// Mitsubishi GX Developer project: 粗材ストッカー   PLC: Q02

PROGRAM MAIN
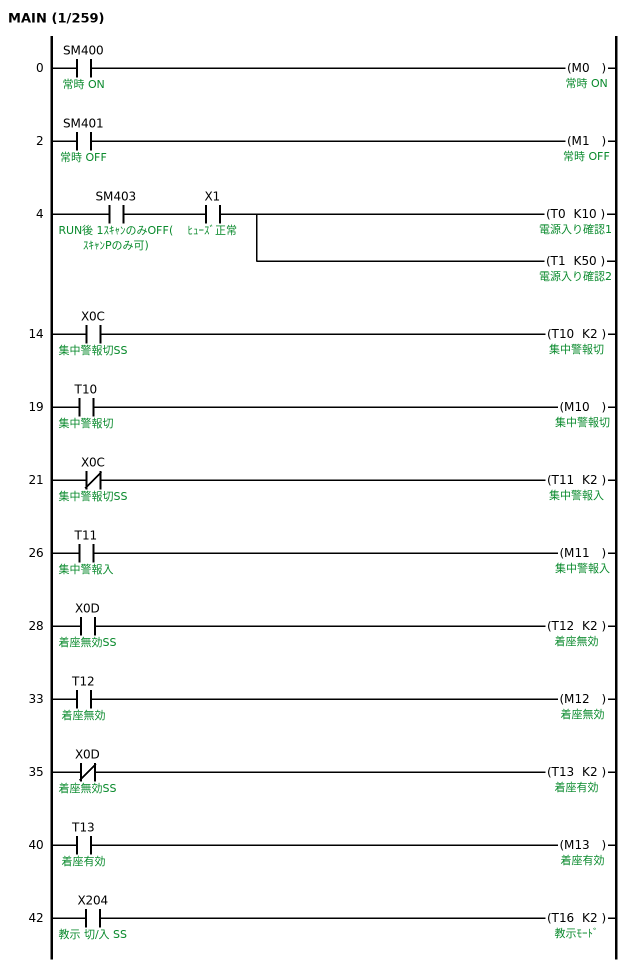
0     LD      SM400  ; 常時 ON
      OUT     M0  ; 常時 ON
2     LD      SM401  ; 常時 OFF
      OUT     M1  ; 常時 OFF
4     LD      SM403  ; RUN後 1ｽｷｬﾝのみOFF(ｽｷｬﾝPのみ可)
      AND     X1  ; ﾋｭｰｽﾞ正常
      OUT     T0 K10  ; 電源入り確認1
      OUT     T1 K50  ; 電源入り確認2
14    LD      X0C  ; 集中警報切SS
      OUT     T10 K2  ; 集中警報切
19    LD      T10  ; 集中警報切
      OUT     M10  ; 集中警報切
21    LDI     X0C  ; 集中警報切SS
      OUT     T11 K2  ; 集中警報入
26    LD      T11  ; 集中警報入
      OUT     M11  ; 集中警報入
28    LD      X0D  ; 着座無効SS
      OUT     T12 K2  ; 着座無効
33    LD      T12  ; 着座無効
      OUT     M12  ; 着座無効
35    LDI     X0D  ; 着座無効SS
      OUT     T13 K2  ; 着座有効
40    LD      T13  ; 着座有効
      OUT     M13  ; 着座有効
42    LD      X204  ; 教示 切/入 SS
      OUT     T16 K2  ; 教示ﾓｰﾄﾞ
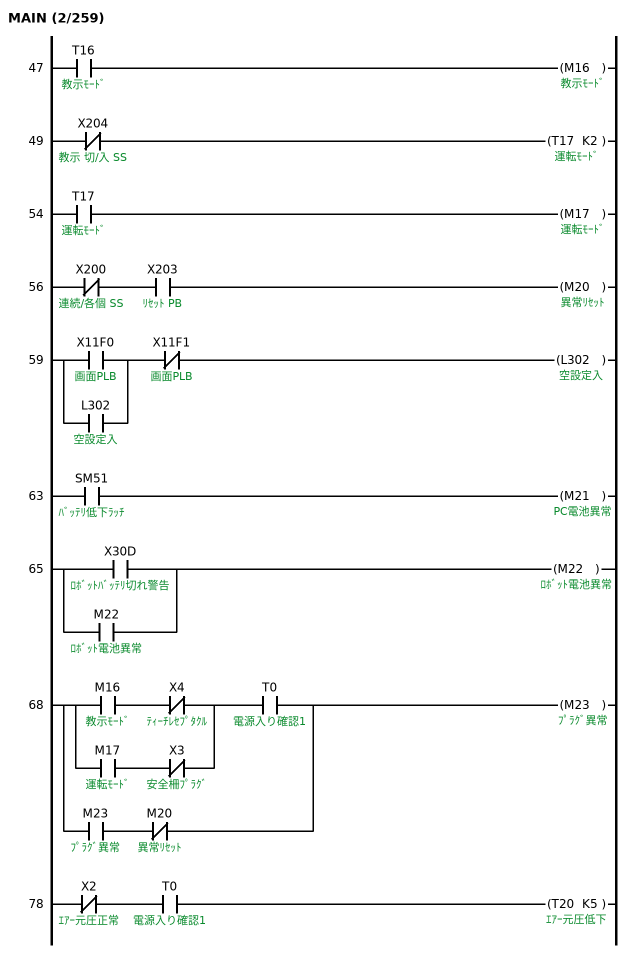
47    LD      T16  ; 教示ﾓｰﾄﾞ
      OUT     M16  ; 教示ﾓｰﾄﾞ
49    LDI     X204  ; 教示 切/入 SS
      OUT     T17 K2  ; 運転ﾓｰﾄﾞ
54    LD      T17  ; 運転ﾓｰﾄﾞ
      OUT     M17  ; 運転ﾓｰﾄﾞ
56    LDI     X200  ; 連続/各個 SS
      AND     X203  ; ﾘｾｯﾄ PB
      OUT     M20  ; 異常ﾘｾｯﾄ
59    LD      X11F0  ; 画面PLB
      OR      L302  ; 空設定入
      ANI     X11F1  ; 画面PLB
      OUT     L302  ; 空設定入
63    LD      SM51  ; ﾊﾞｯﾃﾘ低下ﾗｯﾁ
      OUT     M21  ; PC電池異常
65    LD      X30D  ; ﾛﾎﾞｯﾄﾊﾞｯﾃﾘ切れ警告
      OR      M22  ; ﾛﾎﾞｯﾄ電池異常
      OUT     M22  ; ﾛﾎﾞｯﾄ電池異常
68    LD      M16  ; 教示ﾓｰﾄﾞ
      ANI     X4  ; ﾃｨｰﾁﾚｾﾌﾟﾀｸﾙ
      LD      M17  ; 運転ﾓｰﾄﾞ
      ANI     X3  ; 安全柵ﾌﾟﾗｸﾞ
      ORB
      AND     T0  ; 電源入り確認1
      LD      M23  ; ﾌﾟﾗｸﾞ異常
      ANI     M20  ; 異常ﾘｾｯﾄ
      ORB
      OUT     M23  ; ﾌﾟﾗｸﾞ異常
78    LDI     X2  ; ｴｱｰ元圧正常
      AND     T0  ; 電源入り確認1
      OUT     T20 K5  ; ｴｱｰ元圧低下
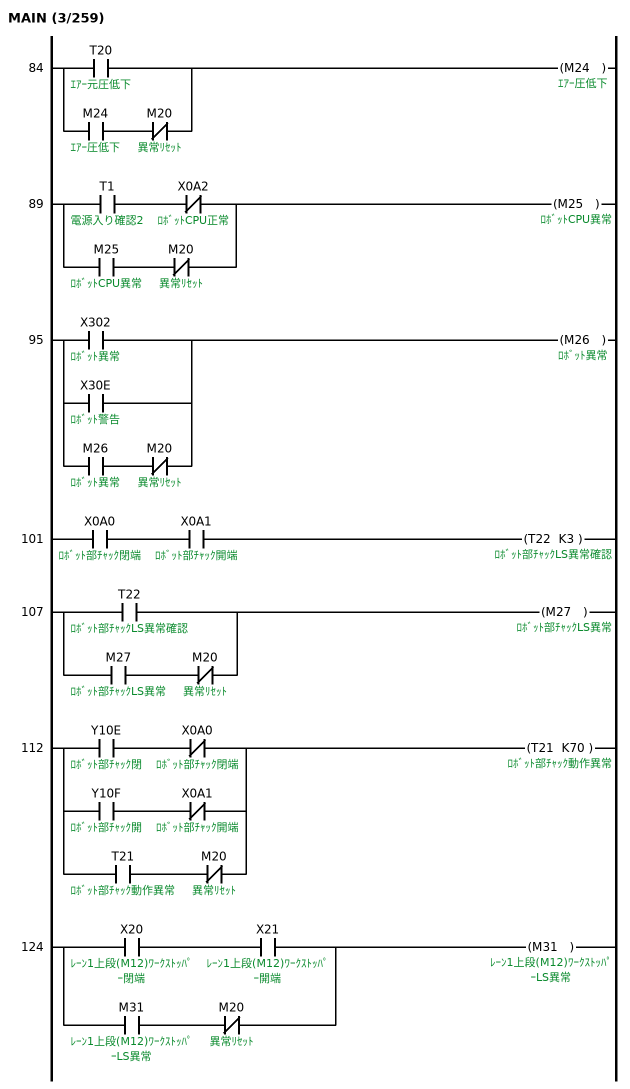
84    LD      T20  ; ｴｱｰ元圧低下
      LD      M24  ; ｴｱｰ圧低下
      ANI     M20  ; 異常ﾘｾｯﾄ
      ORB
      OUT     M24  ; ｴｱｰ圧低下
89    LD      T1  ; 電源入り確認2
      ANI     X0A2  ; ﾛﾎﾞｯﾄCPU正常
      LD      M25  ; ﾛﾎﾞｯﾄCPU異常
      ANI     M20  ; 異常ﾘｾｯﾄ
      ORB
      OUT     M25  ; ﾛﾎﾞｯﾄCPU異常
95    LD      X302  ; ﾛﾎﾞｯﾄ異常
      OR      X30E  ; ﾛﾎﾞｯﾄ警告
      LD      M26  ; ﾛﾎﾞｯﾄ異常
      ANI     M20  ; 異常ﾘｾｯﾄ
      ORB
      OUT     M26  ; ﾛﾎﾞｯﾄ異常
101   LD      X0A0  ; ﾛﾎﾞｯﾄ部ﾁｬｯｸ閉端
      AND     X0A1  ; ﾛﾎﾞｯﾄ部ﾁｬｯｸ開端
      OUT     T22 K3  ; ﾛﾎﾞｯﾄ部ﾁｬｯｸLS異常確認
107   LD      T22  ; ﾛﾎﾞｯﾄ部ﾁｬｯｸLS異常確認
      LD      M27  ; ﾛﾎﾞｯﾄ部ﾁｬｯｸLS異常
      ANI     M20  ; 異常ﾘｾｯﾄ
      ORB
      OUT     M27  ; ﾛﾎﾞｯﾄ部ﾁｬｯｸLS異常
112   LD      Y10E  ; ﾛﾎﾞｯﾄ部ﾁｬｯｸ閉
      ANI     X0A0  ; ﾛﾎﾞｯﾄ部ﾁｬｯｸ閉端
      LD      Y10F  ; ﾛﾎﾞｯﾄ部ﾁｬｯｸ開
      ANI     X0A1  ; ﾛﾎﾞｯﾄ部ﾁｬｯｸ開端
      ORB
      LD      T21  ; ﾛﾎﾞｯﾄ部ﾁｬｯｸ動作異常
      ANI     M20  ; 異常ﾘｾｯﾄ
      ORB
      OUT     T21 K70  ; ﾛﾎﾞｯﾄ部ﾁｬｯｸ動作異常
124   LD      X20  ; ﾚｰﾝ1上段(M12)ﾜｰｸｽﾄｯﾊﾟｰ閉端
      AND     X21  ; ﾚｰﾝ1上段(M12)ﾜｰｸｽﾄｯﾊﾟｰ開端
      LD      M31  ; ﾚｰﾝ1上段(M12)ﾜｰｸｽﾄｯﾊﾟｰLS異常
      ANI     M20  ; 異常ﾘｾｯﾄ
      ORB
      OUT     M31  ; ﾚｰﾝ1上段(M12)ﾜｰｸｽﾄｯﾊﾟｰLS異常
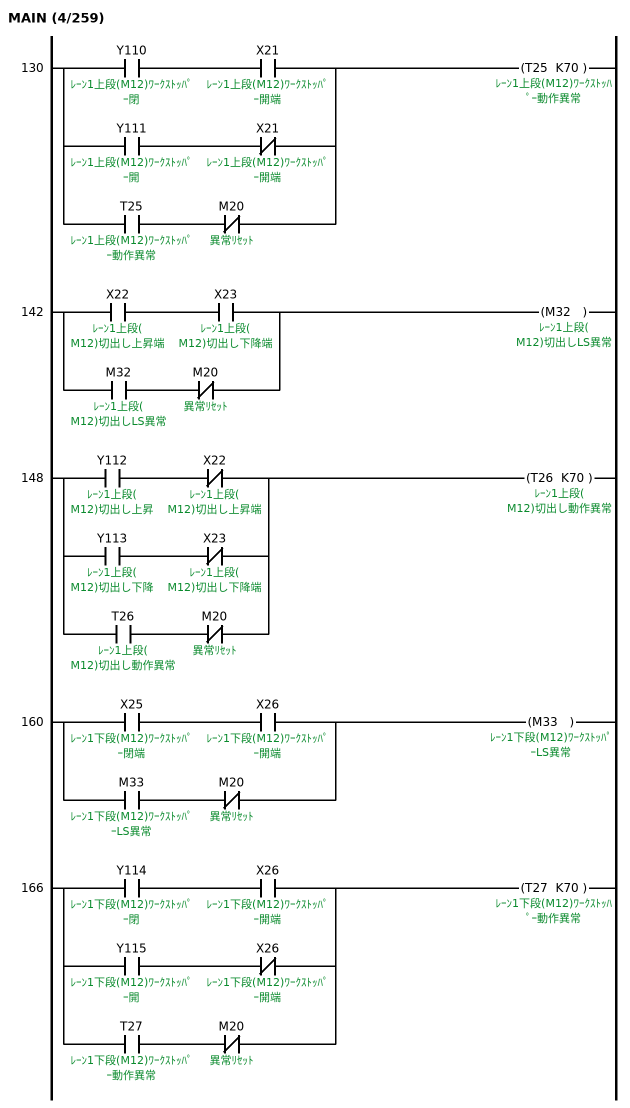
130   LD      Y110  ; ﾚｰﾝ1上段(M12)ﾜｰｸｽﾄｯﾊﾟｰ閉
      AND     X21  ; ﾚｰﾝ1上段(M12)ﾜｰｸｽﾄｯﾊﾟｰ開端
      LD      Y111  ; ﾚｰﾝ1上段(M12)ﾜｰｸｽﾄｯﾊﾟｰ開
      ANI     X21  ; ﾚｰﾝ1上段(M12)ﾜｰｸｽﾄｯﾊﾟｰ開端
      ORB
      LD      T25  ; ﾚｰﾝ1上段(M12)ﾜｰｸｽﾄｯﾊﾟｰ動作異常
      ANI     M20  ; 異常ﾘｾｯﾄ
      ORB
      OUT     T25 K70  ; ﾚｰﾝ1上段(M12)ﾜｰｸｽﾄｯﾊﾟｰ動作異常
142   LD      X22  ; ﾚｰﾝ1上段(M12)切出し上昇端
      AND     X23  ; ﾚｰﾝ1上段(M12)切出し下降端
      LD      M32  ; ﾚｰﾝ1上段(M12)切出しLS異常
      ANI     M20  ; 異常ﾘｾｯﾄ
      ORB
      OUT     M32  ; ﾚｰﾝ1上段(M12)切出しLS異常
148   LD      Y112  ; ﾚｰﾝ1上段(M12)切出し上昇
      ANI     X22  ; ﾚｰﾝ1上段(M12)切出し上昇端
      LD      Y113  ; ﾚｰﾝ1上段(M12)切出し下降
      ANI     X23  ; ﾚｰﾝ1上段(M12)切出し下降端
      ORB
      LD      T26  ; ﾚｰﾝ1上段(M12)切出し動作異常
      ANI     M20  ; 異常ﾘｾｯﾄ
      ORB
      OUT     T26 K70  ; ﾚｰﾝ1上段(M12)切出し動作異常
160   LD      X25  ; ﾚｰﾝ1下段(M12)ﾜｰｸｽﾄｯﾊﾟｰ閉端
      AND     X26  ; ﾚｰﾝ1下段(M12)ﾜｰｸｽﾄｯﾊﾟｰ開端
      LD      M33  ; ﾚｰﾝ1下段(M12)ﾜｰｸｽﾄｯﾊﾟｰLS異常
      ANI     M20  ; 異常ﾘｾｯﾄ
      ORB
      OUT     M33  ; ﾚｰﾝ1下段(M12)ﾜｰｸｽﾄｯﾊﾟｰLS異常
166   LD      Y114  ; ﾚｰﾝ1下段(M12)ﾜｰｸｽﾄｯﾊﾟｰ閉
      AND     X26  ; ﾚｰﾝ1下段(M12)ﾜｰｸｽﾄｯﾊﾟｰ開端
      LD      Y115  ; ﾚｰﾝ1下段(M12)ﾜｰｸｽﾄｯﾊﾟｰ開
      ANI     X26  ; ﾚｰﾝ1下段(M12)ﾜｰｸｽﾄｯﾊﾟｰ開端
      ORB
      LD      T27  ; ﾚｰﾝ1下段(M12)ﾜｰｸｽﾄｯﾊﾟｰ動作異常
      ANI     M20  ; 異常ﾘｾｯﾄ
      ORB
      OUT     T27 K70  ; ﾚｰﾝ1下段(M12)ﾜｰｸｽﾄｯﾊﾟｰ動作異常
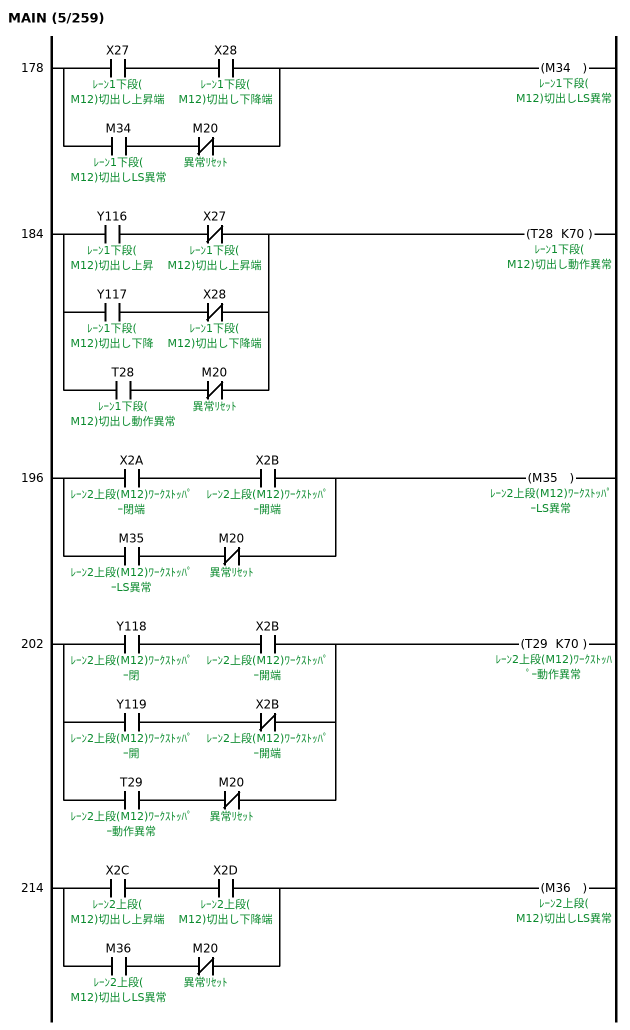
178   LD      X27  ; ﾚｰﾝ1下段(M12)切出し上昇端
      AND     X28  ; ﾚｰﾝ1下段(M12)切出し下降端
      LD      M34  ; ﾚｰﾝ1下段(M12)切出しLS異常
      ANI     M20  ; 異常ﾘｾｯﾄ
      ORB
      OUT     M34  ; ﾚｰﾝ1下段(M12)切出しLS異常
184   LD      Y116  ; ﾚｰﾝ1下段(M12)切出し上昇
      ANI     X27  ; ﾚｰﾝ1下段(M12)切出し上昇端
      LD      Y117  ; ﾚｰﾝ1下段(M12)切出し下降
      ANI     X28  ; ﾚｰﾝ1下段(M12)切出し下降端
      ORB
      LD      T28  ; ﾚｰﾝ1下段(M12)切出し動作異常
      ANI     M20  ; 異常ﾘｾｯﾄ
      ORB
      OUT     T28 K70  ; ﾚｰﾝ1下段(M12)切出し動作異常
196   LD      X2A  ; ﾚｰﾝ2上段(M12)ﾜｰｸｽﾄｯﾊﾟｰ閉端
      AND     X2B  ; ﾚｰﾝ2上段(M12)ﾜｰｸｽﾄｯﾊﾟｰ開端
      LD      M35  ; ﾚｰﾝ2上段(M12)ﾜｰｸｽﾄｯﾊﾟｰLS異常
      ANI     M20  ; 異常ﾘｾｯﾄ
      ORB
      OUT     M35  ; ﾚｰﾝ2上段(M12)ﾜｰｸｽﾄｯﾊﾟｰLS異常
202   LD      Y118  ; ﾚｰﾝ2上段(M12)ﾜｰｸｽﾄｯﾊﾟｰ閉
      AND     X2B  ; ﾚｰﾝ2上段(M12)ﾜｰｸｽﾄｯﾊﾟｰ開端
      LD      Y119  ; ﾚｰﾝ2上段(M12)ﾜｰｸｽﾄｯﾊﾟｰ開
      ANI     X2B  ; ﾚｰﾝ2上段(M12)ﾜｰｸｽﾄｯﾊﾟｰ開端
      ORB
      LD      T29  ; ﾚｰﾝ2上段(M12)ﾜｰｸｽﾄｯﾊﾟｰ動作異常
      ANI     M20  ; 異常ﾘｾｯﾄ
      ORB
      OUT     T29 K70  ; ﾚｰﾝ2上段(M12)ﾜｰｸｽﾄｯﾊﾟｰ動作異常
214   LD      X2C  ; ﾚｰﾝ2上段(M12)切出し上昇端
      AND     X2D  ; ﾚｰﾝ2上段(M12)切出し下降端
      LD      M36  ; ﾚｰﾝ2上段(M12)切出しLS異常
      ANI     M20  ; 異常ﾘｾｯﾄ
      ORB
      OUT     M36  ; ﾚｰﾝ2上段(M12)切出しLS異常
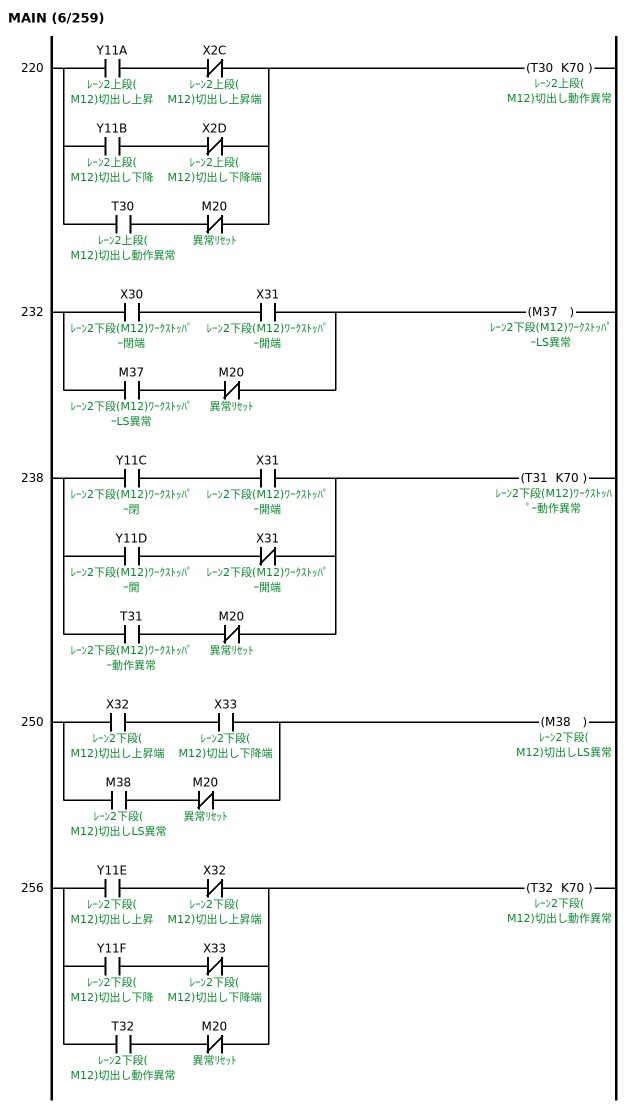
220   LD      Y11A  ; ﾚｰﾝ2上段(M12)切出し上昇
      ANI     X2C  ; ﾚｰﾝ2上段(M12)切出し上昇端
      LD      Y11B  ; ﾚｰﾝ2上段(M12)切出し下降
      ANI     X2D  ; ﾚｰﾝ2上段(M12)切出し下降端
      ORB
      LD      T30  ; ﾚｰﾝ2上段(M12)切出し動作異常
      ANI     M20  ; 異常ﾘｾｯﾄ
      ORB
      OUT     T30 K70  ; ﾚｰﾝ2上段(M12)切出し動作異常
232   LD      X30  ; ﾚｰﾝ2下段(M12)ﾜｰｸｽﾄｯﾊﾟｰ閉端
      AND     X31  ; ﾚｰﾝ2下段(M12)ﾜｰｸｽﾄｯﾊﾟｰ開端
      LD      M37  ; ﾚｰﾝ2下段(M12)ﾜｰｸｽﾄｯﾊﾟｰLS異常
      ANI     M20  ; 異常ﾘｾｯﾄ
      ORB
      OUT     M37  ; ﾚｰﾝ2下段(M12)ﾜｰｸｽﾄｯﾊﾟｰLS異常
238   LD      Y11C  ; ﾚｰﾝ2下段(M12)ﾜｰｸｽﾄｯﾊﾟｰ閉
      AND     X31  ; ﾚｰﾝ2下段(M12)ﾜｰｸｽﾄｯﾊﾟｰ開端
      LD      Y11D  ; ﾚｰﾝ2下段(M12)ﾜｰｸｽﾄｯﾊﾟｰ開
      ANI     X31  ; ﾚｰﾝ2下段(M12)ﾜｰｸｽﾄｯﾊﾟｰ開端
      ORB
      LD      T31  ; ﾚｰﾝ2下段(M12)ﾜｰｸｽﾄｯﾊﾟｰ動作異常
      ANI     M20  ; 異常ﾘｾｯﾄ
      ORB
      OUT     T31 K70  ; ﾚｰﾝ2下段(M12)ﾜｰｸｽﾄｯﾊﾟｰ動作異常
250   LD      X32  ; ﾚｰﾝ2下段(M12)切出し上昇端
      AND     X33  ; ﾚｰﾝ2下段(M12)切出し下降端
      LD      M38  ; ﾚｰﾝ2下段(M12)切出しLS異常
      ANI     M20  ; 異常ﾘｾｯﾄ
      ORB
      OUT     M38  ; ﾚｰﾝ2下段(M12)切出しLS異常
256   LD      Y11E  ; ﾚｰﾝ2下段(M12)切出し上昇
      ANI     X32  ; ﾚｰﾝ2下段(M12)切出し上昇端
      LD      Y11F  ; ﾚｰﾝ2下段(M12)切出し下降
      ANI     X33  ; ﾚｰﾝ2下段(M12)切出し下降端
      ORB
      LD      T32  ; ﾚｰﾝ2下段(M12)切出し動作異常
      ANI     M20  ; 異常ﾘｾｯﾄ
      ORB
      OUT     T32 K70  ; ﾚｰﾝ2下段(M12)切出し動作異常
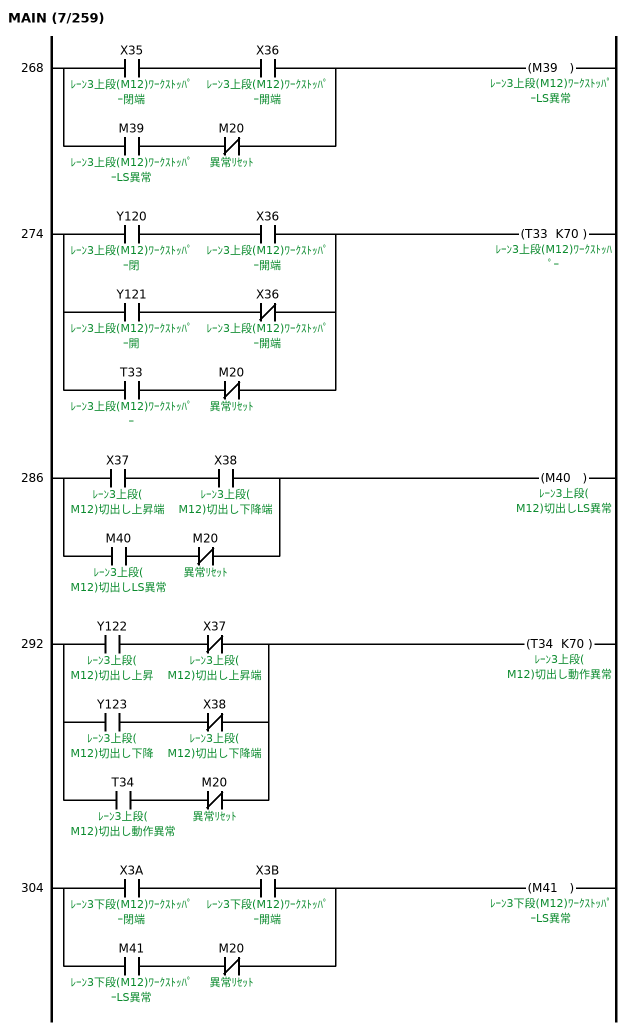
268   LD      X35  ; ﾚｰﾝ3上段(M12)ﾜｰｸｽﾄｯﾊﾟｰ閉端
      AND     X36  ; ﾚｰﾝ3上段(M12)ﾜｰｸｽﾄｯﾊﾟｰ開端
      LD      M39  ; ﾚｰﾝ3上段(M12)ﾜｰｸｽﾄｯﾊﾟｰLS異常
      ANI     M20  ; 異常ﾘｾｯﾄ
      ORB
      OUT     M39  ; ﾚｰﾝ3上段(M12)ﾜｰｸｽﾄｯﾊﾟｰLS異常
274   LD      Y120  ; ﾚｰﾝ3上段(M12)ﾜｰｸｽﾄｯﾊﾟｰ閉
      AND     X36  ; ﾚｰﾝ3上段(M12)ﾜｰｸｽﾄｯﾊﾟｰ開端
      LD      Y121  ; ﾚｰﾝ3上段(M12)ﾜｰｸｽﾄｯﾊﾟｰ開
      ANI     X36  ; ﾚｰﾝ3上段(M12)ﾜｰｸｽﾄｯﾊﾟｰ開端
      ORB
      LD      T33  ; ﾚｰﾝ3上段(M12)ﾜｰｸｽﾄｯﾊﾟｰ
      ANI     M20  ; 異常ﾘｾｯﾄ
      ORB
      OUT     T33 K70  ; ﾚｰﾝ3上段(M12)ﾜｰｸｽﾄｯﾊﾟｰ
286   LD      X37  ; ﾚｰﾝ3上段(M12)切出し上昇端
      AND     X38  ; ﾚｰﾝ3上段(M12)切出し下降端
      LD      M40  ; ﾚｰﾝ3上段(M12)切出しLS異常
      ANI     M20  ; 異常ﾘｾｯﾄ
      ORB
      OUT     M40  ; ﾚｰﾝ3上段(M12)切出しLS異常
292   LD      Y122  ; ﾚｰﾝ3上段(M12)切出し上昇
      ANI     X37  ; ﾚｰﾝ3上段(M12)切出し上昇端
      LD      Y123  ; ﾚｰﾝ3上段(M12)切出し下降
      ANI     X38  ; ﾚｰﾝ3上段(M12)切出し下降端
      ORB
      LD      T34  ; ﾚｰﾝ3上段(M12)切出し動作異常
      ANI     M20  ; 異常ﾘｾｯﾄ
      ORB
      OUT     T34 K70  ; ﾚｰﾝ3上段(M12)切出し動作異常
304   LD      X3A  ; ﾚｰﾝ3下段(M12)ﾜｰｸｽﾄｯﾊﾟｰ閉端
      AND     X3B  ; ﾚｰﾝ3下段(M12)ﾜｰｸｽﾄｯﾊﾟｰ開端
      LD      M41  ; ﾚｰﾝ3下段(M12)ﾜｰｸｽﾄｯﾊﾟｰLS異常
      ANI     M20  ; 異常ﾘｾｯﾄ
      ORB
      OUT     M41  ; ﾚｰﾝ3下段(M12)ﾜｰｸｽﾄｯﾊﾟｰLS異常
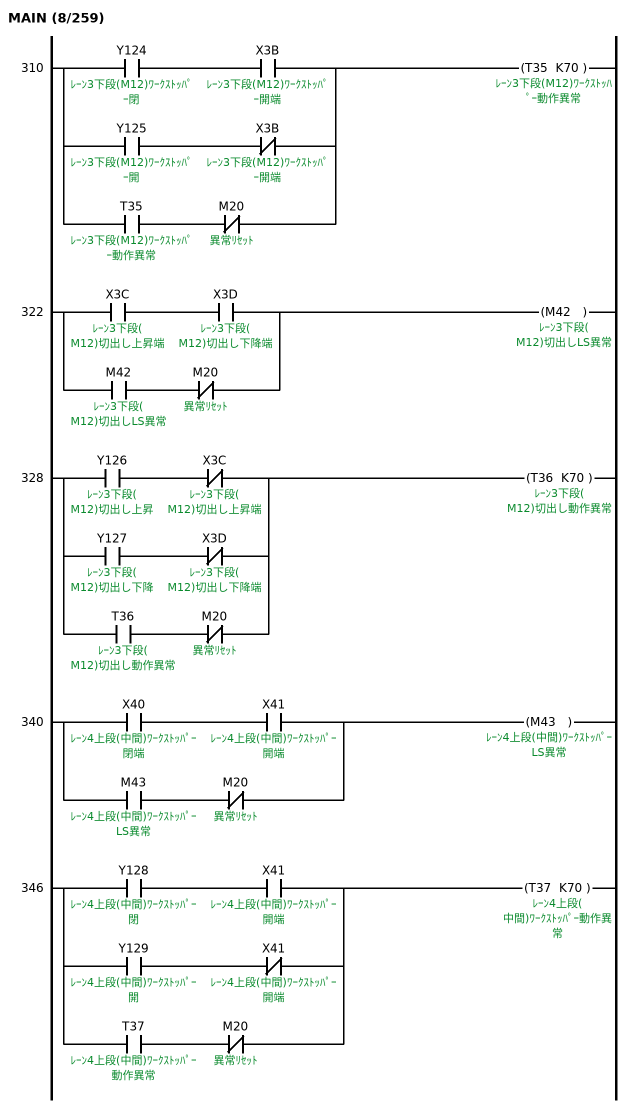
310   LD      Y124  ; ﾚｰﾝ3下段(M12)ﾜｰｸｽﾄｯﾊﾟｰ閉
      AND     X3B  ; ﾚｰﾝ3下段(M12)ﾜｰｸｽﾄｯﾊﾟｰ開端
      LD      Y125  ; ﾚｰﾝ3下段(M12)ﾜｰｸｽﾄｯﾊﾟｰ開
      ANI     X3B  ; ﾚｰﾝ3下段(M12)ﾜｰｸｽﾄｯﾊﾟｰ開端
      ORB
      LD      T35  ; ﾚｰﾝ3下段(M12)ﾜｰｸｽﾄｯﾊﾟｰ動作異常
      ANI     M20  ; 異常ﾘｾｯﾄ
      ORB
      OUT     T35 K70  ; ﾚｰﾝ3下段(M12)ﾜｰｸｽﾄｯﾊﾟｰ動作異常
322   LD      X3C  ; ﾚｰﾝ3下段(M12)切出し上昇端
      AND     X3D  ; ﾚｰﾝ3下段(M12)切出し下降端
      LD      M42  ; ﾚｰﾝ3下段(M12)切出しLS異常
      ANI     M20  ; 異常ﾘｾｯﾄ
      ORB
      OUT     M42  ; ﾚｰﾝ3下段(M12)切出しLS異常
328   LD      Y126  ; ﾚｰﾝ3下段(M12)切出し上昇
      ANI     X3C  ; ﾚｰﾝ3下段(M12)切出し上昇端
      LD      Y127  ; ﾚｰﾝ3下段(M12)切出し下降
      ANI     X3D  ; ﾚｰﾝ3下段(M12)切出し下降端
      ORB
      LD      T36  ; ﾚｰﾝ3下段(M12)切出し動作異常
      ANI     M20  ; 異常ﾘｾｯﾄ
      ORB
      OUT     T36 K70  ; ﾚｰﾝ3下段(M12)切出し動作異常
340   LD      X40  ; ﾚｰﾝ4上段(中間)ﾜｰｸｽﾄｯﾊﾟｰ閉端
      AND     X41  ; ﾚｰﾝ4上段(中間)ﾜｰｸｽﾄｯﾊﾟｰ開端
      LD      M43  ; ﾚｰﾝ4上段(中間)ﾜｰｸｽﾄｯﾊﾟｰLS異常
      ANI     M20  ; 異常ﾘｾｯﾄ
      ORB
      OUT     M43  ; ﾚｰﾝ4上段(中間)ﾜｰｸｽﾄｯﾊﾟｰLS異常
346   LD      Y128  ; ﾚｰﾝ4上段(中間)ﾜｰｸｽﾄｯﾊﾟｰ閉
      AND     X41  ; ﾚｰﾝ4上段(中間)ﾜｰｸｽﾄｯﾊﾟｰ開端
      LD      Y129  ; ﾚｰﾝ4上段(中間)ﾜｰｸｽﾄｯﾊﾟｰ開
      ANI     X41  ; ﾚｰﾝ4上段(中間)ﾜｰｸｽﾄｯﾊﾟｰ開端
      ORB
      LD      T37  ; ﾚｰﾝ4上段(中間)ﾜｰｸｽﾄｯﾊﾟｰ動作異常
      ANI     M20  ; 異常ﾘｾｯﾄ
      ORB
      OUT     T37 K70  ; ﾚｰﾝ4上段(中間)ﾜｰｸｽﾄｯﾊﾟｰ動作異常
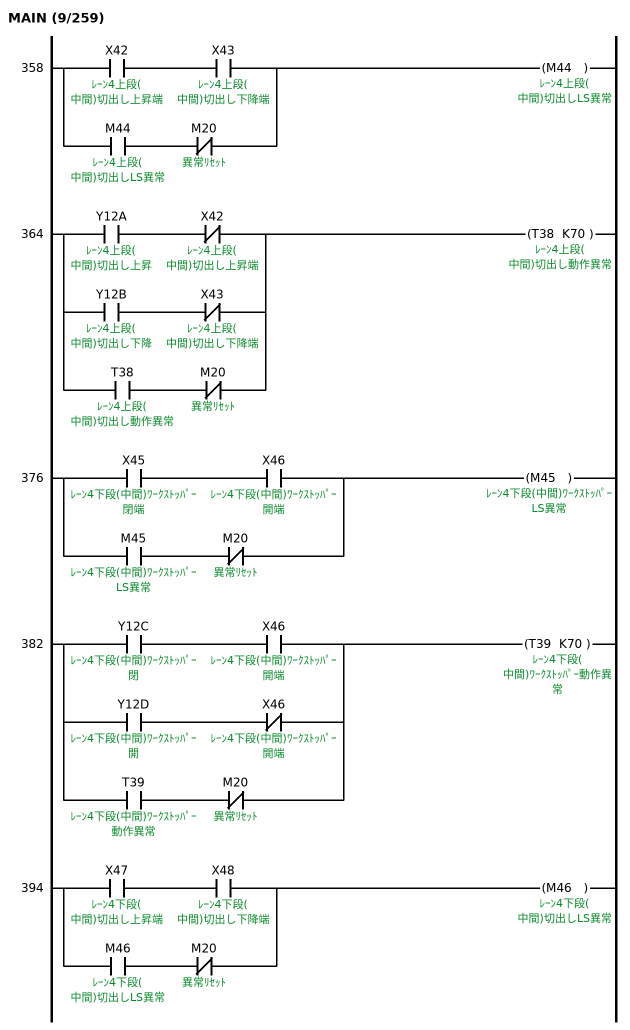
358   LD      X42  ; ﾚｰﾝ4上段(中間)切出し上昇端
      AND     X43  ; ﾚｰﾝ4上段(中間)切出し下降端
      LD      M44  ; ﾚｰﾝ4上段(中間)切出しLS異常
      ANI     M20  ; 異常ﾘｾｯﾄ
      ORB
      OUT     M44  ; ﾚｰﾝ4上段(中間)切出しLS異常
364   LD      Y12A  ; ﾚｰﾝ4上段(中間)切出し上昇
      ANI     X42  ; ﾚｰﾝ4上段(中間)切出し上昇端
      LD      Y12B  ; ﾚｰﾝ4上段(中間)切出し下降
      ANI     X43  ; ﾚｰﾝ4上段(中間)切出し下降端
      ORB
      LD      T38  ; ﾚｰﾝ4上段(中間)切出し動作異常
      ANI     M20  ; 異常ﾘｾｯﾄ
      ORB
      OUT     T38 K70  ; ﾚｰﾝ4上段(中間)切出し動作異常
376   LD      X45  ; ﾚｰﾝ4下段(中間)ﾜｰｸｽﾄｯﾊﾟｰ閉端
      AND     X46  ; ﾚｰﾝ4下段(中間)ﾜｰｸｽﾄｯﾊﾟｰ開端
      LD      M45  ; ﾚｰﾝ4下段(中間)ﾜｰｸｽﾄｯﾊﾟｰLS異常
      ANI     M20  ; 異常ﾘｾｯﾄ
      ORB
      OUT     M45  ; ﾚｰﾝ4下段(中間)ﾜｰｸｽﾄｯﾊﾟｰLS異常
382   LD      Y12C  ; ﾚｰﾝ4下段(中間)ﾜｰｸｽﾄｯﾊﾟｰ閉
      AND     X46  ; ﾚｰﾝ4下段(中間)ﾜｰｸｽﾄｯﾊﾟｰ開端
      LD      Y12D  ; ﾚｰﾝ4下段(中間)ﾜｰｸｽﾄｯﾊﾟｰ開
      ANI     X46  ; ﾚｰﾝ4下段(中間)ﾜｰｸｽﾄｯﾊﾟｰ開端
      ORB
      LD      T39  ; ﾚｰﾝ4下段(中間)ﾜｰｸｽﾄｯﾊﾟｰ動作異常
      ANI     M20  ; 異常ﾘｾｯﾄ
      ORB
      OUT     T39 K70  ; ﾚｰﾝ4下段(中間)ﾜｰｸｽﾄｯﾊﾟｰ動作異常
394   LD      X47  ; ﾚｰﾝ4下段(中間)切出し上昇端
      AND     X48  ; ﾚｰﾝ4下段(中間)切出し下降端
      LD      M46  ; ﾚｰﾝ4下段(中間)切出しLS異常
      ANI     M20  ; 異常ﾘｾｯﾄ
      ORB
      OUT     M46  ; ﾚｰﾝ4下段(中間)切出しLS異常
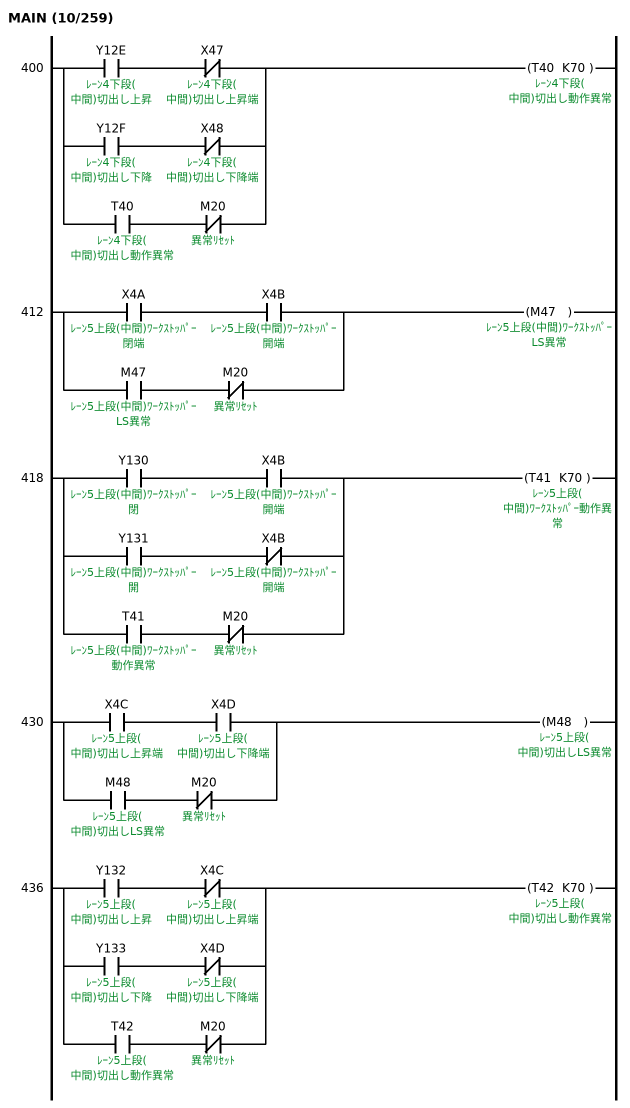
400   LD      Y12E  ; ﾚｰﾝ4下段(中間)切出し上昇
      ANI     X47  ; ﾚｰﾝ4下段(中間)切出し上昇端
      LD      Y12F  ; ﾚｰﾝ4下段(中間)切出し下降
      ANI     X48  ; ﾚｰﾝ4下段(中間)切出し下降端
      ORB
      LD      T40  ; ﾚｰﾝ4下段(中間)切出し動作異常
      ANI     M20  ; 異常ﾘｾｯﾄ
      ORB
      OUT     T40 K70  ; ﾚｰﾝ4下段(中間)切出し動作異常
412   LD      X4A  ; ﾚｰﾝ5上段(中間)ﾜｰｸｽﾄｯﾊﾟｰ閉端
      AND     X4B  ; ﾚｰﾝ5上段(中間)ﾜｰｸｽﾄｯﾊﾟｰ開端
      LD      M47  ; ﾚｰﾝ5上段(中間)ﾜｰｸｽﾄｯﾊﾟｰLS異常
      ANI     M20  ; 異常ﾘｾｯﾄ
      ORB
      OUT     M47  ; ﾚｰﾝ5上段(中間)ﾜｰｸｽﾄｯﾊﾟｰLS異常
418   LD      Y130  ; ﾚｰﾝ5上段(中間)ﾜｰｸｽﾄｯﾊﾟｰ閉
      AND     X4B  ; ﾚｰﾝ5上段(中間)ﾜｰｸｽﾄｯﾊﾟｰ開端
      LD      Y131  ; ﾚｰﾝ5上段(中間)ﾜｰｸｽﾄｯﾊﾟｰ開
      ANI     X4B  ; ﾚｰﾝ5上段(中間)ﾜｰｸｽﾄｯﾊﾟｰ開端
      ORB
      LD      T41  ; ﾚｰﾝ5上段(中間)ﾜｰｸｽﾄｯﾊﾟｰ動作異常
      ANI     M20  ; 異常ﾘｾｯﾄ
      ORB
      OUT     T41 K70  ; ﾚｰﾝ5上段(中間)ﾜｰｸｽﾄｯﾊﾟｰ動作異常
430   LD      X4C  ; ﾚｰﾝ5上段(中間)切出し上昇端
      AND     X4D  ; ﾚｰﾝ5上段(中間)切出し下降端
      LD      M48  ; ﾚｰﾝ5上段(中間)切出しLS異常
      ANI     M20  ; 異常ﾘｾｯﾄ
      ORB
      OUT     M48  ; ﾚｰﾝ5上段(中間)切出しLS異常
436   LD      Y132  ; ﾚｰﾝ5上段(中間)切出し上昇
      ANI     X4C  ; ﾚｰﾝ5上段(中間)切出し上昇端
      LD      Y133  ; ﾚｰﾝ5上段(中間)切出し下降
      ANI     X4D  ; ﾚｰﾝ5上段(中間)切出し下降端
      ORB
      LD      T42  ; ﾚｰﾝ5上段(中間)切出し動作異常
      ANI     M20  ; 異常ﾘｾｯﾄ
      ORB
      OUT     T42 K70  ; ﾚｰﾝ5上段(中間)切出し動作異常
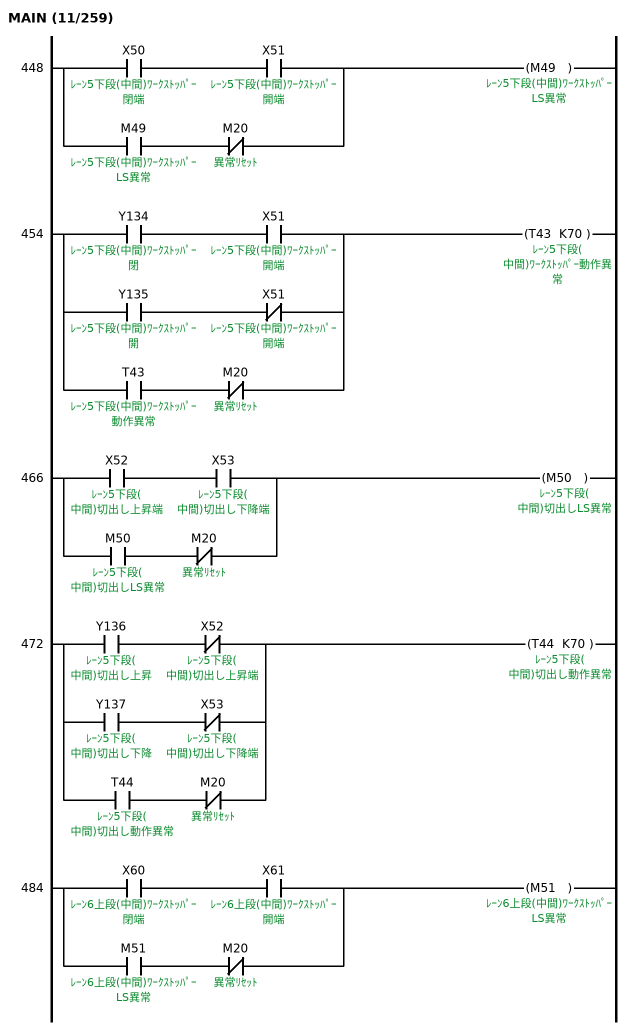
448   LD      X50  ; ﾚｰﾝ5下段(中間)ﾜｰｸｽﾄｯﾊﾟｰ閉端
      AND     X51  ; ﾚｰﾝ5下段(中間)ﾜｰｸｽﾄｯﾊﾟｰ開端
      LD      M49  ; ﾚｰﾝ5下段(中間)ﾜｰｸｽﾄｯﾊﾟｰLS異常
      ANI     M20  ; 異常ﾘｾｯﾄ
      ORB
      OUT     M49  ; ﾚｰﾝ5下段(中間)ﾜｰｸｽﾄｯﾊﾟｰLS異常
454   LD      Y134  ; ﾚｰﾝ5下段(中間)ﾜｰｸｽﾄｯﾊﾟｰ閉
      AND     X51  ; ﾚｰﾝ5下段(中間)ﾜｰｸｽﾄｯﾊﾟｰ開端
      LD      Y135  ; ﾚｰﾝ5下段(中間)ﾜｰｸｽﾄｯﾊﾟｰ開
      ANI     X51  ; ﾚｰﾝ5下段(中間)ﾜｰｸｽﾄｯﾊﾟｰ開端
      ORB
      LD      T43  ; ﾚｰﾝ5下段(中間)ﾜｰｸｽﾄｯﾊﾟｰ動作異常
      ANI     M20  ; 異常ﾘｾｯﾄ
      ORB
      OUT     T43 K70  ; ﾚｰﾝ5下段(中間)ﾜｰｸｽﾄｯﾊﾟｰ動作異常
466   LD      X52  ; ﾚｰﾝ5下段(中間)切出し上昇端
      AND     X53  ; ﾚｰﾝ5下段(中間)切出し下降端
      LD      M50  ; ﾚｰﾝ5下段(中間)切出しLS異常
      ANI     M20  ; 異常ﾘｾｯﾄ
      ORB
      OUT     M50  ; ﾚｰﾝ5下段(中間)切出しLS異常
472   LD      Y136  ; ﾚｰﾝ5下段(中間)切出し上昇
      ANI     X52  ; ﾚｰﾝ5下段(中間)切出し上昇端
      LD      Y137  ; ﾚｰﾝ5下段(中間)切出し下降
      ANI     X53  ; ﾚｰﾝ5下段(中間)切出し下降端
      ORB
      LD      T44  ; ﾚｰﾝ5下段(中間)切出し動作異常
      ANI     M20  ; 異常ﾘｾｯﾄ
      ORB
      OUT     T44 K70  ; ﾚｰﾝ5下段(中間)切出し動作異常
484   LD      X60  ; ﾚｰﾝ6上段(中間)ﾜｰｸｽﾄｯﾊﾟｰ閉端
      AND     X61  ; ﾚｰﾝ6上段(中間)ﾜｰｸｽﾄｯﾊﾟｰ開端
      LD      M51  ; ﾚｰﾝ6上段(中間)ﾜｰｸｽﾄｯﾊﾟｰLS異常
      ANI     M20  ; 異常ﾘｾｯﾄ
      ORB
      OUT     M51  ; ﾚｰﾝ6上段(中間)ﾜｰｸｽﾄｯﾊﾟｰLS異常
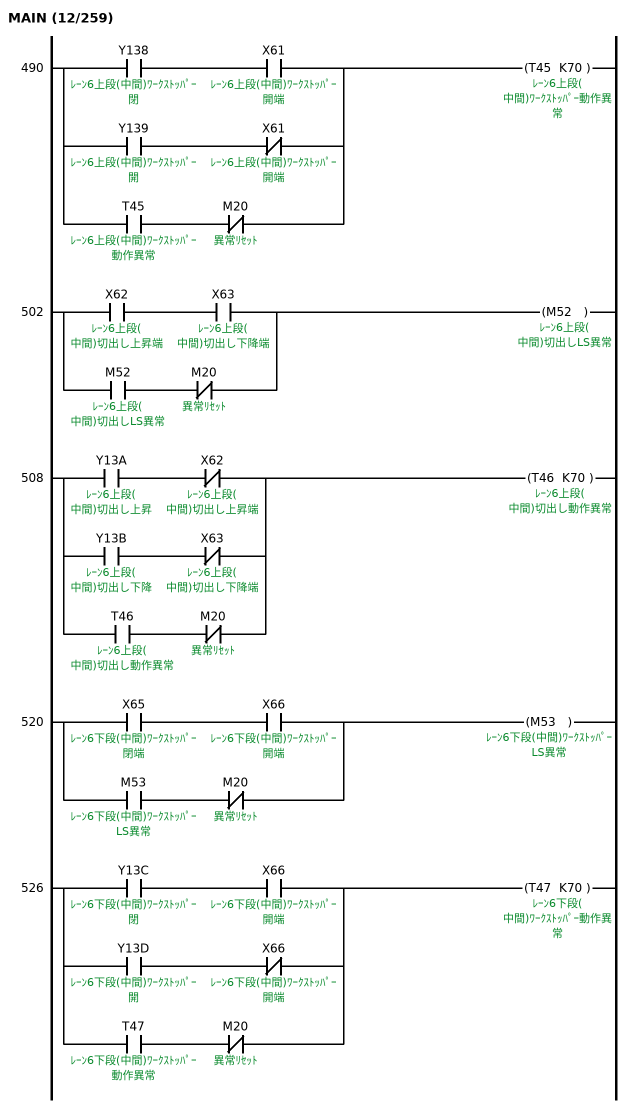
490   LD      Y138  ; ﾚｰﾝ6上段(中間)ﾜｰｸｽﾄｯﾊﾟｰ閉
      AND     X61  ; ﾚｰﾝ6上段(中間)ﾜｰｸｽﾄｯﾊﾟｰ開端
      LD      Y139  ; ﾚｰﾝ6上段(中間)ﾜｰｸｽﾄｯﾊﾟｰ開
      ANI     X61  ; ﾚｰﾝ6上段(中間)ﾜｰｸｽﾄｯﾊﾟｰ開端
      ORB
      LD      T45  ; ﾚｰﾝ6上段(中間)ﾜｰｸｽﾄｯﾊﾟｰ動作異常
      ANI     M20  ; 異常ﾘｾｯﾄ
      ORB
      OUT     T45 K70  ; ﾚｰﾝ6上段(中間)ﾜｰｸｽﾄｯﾊﾟｰ動作異常
502   LD      X62  ; ﾚｰﾝ6上段(中間)切出し上昇端
      AND     X63  ; ﾚｰﾝ6上段(中間)切出し下降端
      LD      M52  ; ﾚｰﾝ6上段(中間)切出しLS異常
      ANI     M20  ; 異常ﾘｾｯﾄ
      ORB
      OUT     M52  ; ﾚｰﾝ6上段(中間)切出しLS異常
508   LD      Y13A  ; ﾚｰﾝ6上段(中間)切出し上昇
      ANI     X62  ; ﾚｰﾝ6上段(中間)切出し上昇端
      LD      Y13B  ; ﾚｰﾝ6上段(中間)切出し下降
      ANI     X63  ; ﾚｰﾝ6上段(中間)切出し下降端
      ORB
      LD      T46  ; ﾚｰﾝ6上段(中間)切出し動作異常
      ANI     M20  ; 異常ﾘｾｯﾄ
      ORB
      OUT     T46 K70  ; ﾚｰﾝ6上段(中間)切出し動作異常
520   LD      X65  ; ﾚｰﾝ6下段(中間)ﾜｰｸｽﾄｯﾊﾟｰ閉端
      AND     X66  ; ﾚｰﾝ6下段(中間)ﾜｰｸｽﾄｯﾊﾟｰ開端
      LD      M53  ; ﾚｰﾝ6下段(中間)ﾜｰｸｽﾄｯﾊﾟｰLS異常
      ANI     M20  ; 異常ﾘｾｯﾄ
      ORB
      OUT     M53  ; ﾚｰﾝ6下段(中間)ﾜｰｸｽﾄｯﾊﾟｰLS異常
526   LD      Y13C  ; ﾚｰﾝ6下段(中間)ﾜｰｸｽﾄｯﾊﾟｰ閉
      AND     X66  ; ﾚｰﾝ6下段(中間)ﾜｰｸｽﾄｯﾊﾟｰ開端
      LD      Y13D  ; ﾚｰﾝ6下段(中間)ﾜｰｸｽﾄｯﾊﾟｰ開
      ANI     X66  ; ﾚｰﾝ6下段(中間)ﾜｰｸｽﾄｯﾊﾟｰ開端
      ORB
      LD      T47  ; ﾚｰﾝ6下段(中間)ﾜｰｸｽﾄｯﾊﾟｰ動作異常
      ANI     M20  ; 異常ﾘｾｯﾄ
      ORB
      OUT     T47 K70  ; ﾚｰﾝ6下段(中間)ﾜｰｸｽﾄｯﾊﾟｰ動作異常
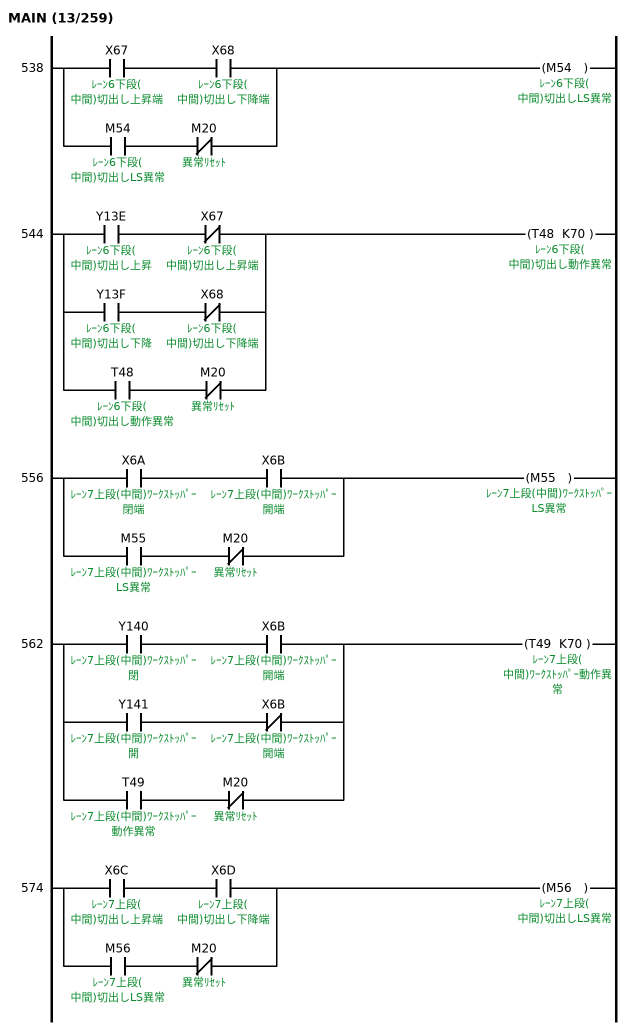
538   LD      X67  ; ﾚｰﾝ6下段(中間)切出し上昇端
      AND     X68  ; ﾚｰﾝ6下段(中間)切出し下降端
      LD      M54  ; ﾚｰﾝ6下段(中間)切出しLS異常
      ANI     M20  ; 異常ﾘｾｯﾄ
      ORB
      OUT     M54  ; ﾚｰﾝ6下段(中間)切出しLS異常
544   LD      Y13E  ; ﾚｰﾝ6下段(中間)切出し上昇
      ANI     X67  ; ﾚｰﾝ6下段(中間)切出し上昇端
      LD      Y13F  ; ﾚｰﾝ6下段(中間)切出し下降
      ANI     X68  ; ﾚｰﾝ6下段(中間)切出し下降端
      ORB
      LD      T48  ; ﾚｰﾝ6下段(中間)切出し動作異常
      ANI     M20  ; 異常ﾘｾｯﾄ
      ORB
      OUT     T48 K70  ; ﾚｰﾝ6下段(中間)切出し動作異常
556   LD      X6A  ; ﾚｰﾝ7上段(中間)ﾜｰｸｽﾄｯﾊﾟｰ閉端
      AND     X6B  ; ﾚｰﾝ7上段(中間)ﾜｰｸｽﾄｯﾊﾟｰ開端
      LD      M55  ; ﾚｰﾝ7上段(中間)ﾜｰｸｽﾄｯﾊﾟｰLS異常
      ANI     M20  ; 異常ﾘｾｯﾄ
      ORB
      OUT     M55  ; ﾚｰﾝ7上段(中間)ﾜｰｸｽﾄｯﾊﾟｰLS異常
562   LD      Y140  ; ﾚｰﾝ7上段(中間)ﾜｰｸｽﾄｯﾊﾟｰ閉
      AND     X6B  ; ﾚｰﾝ7上段(中間)ﾜｰｸｽﾄｯﾊﾟｰ開端
      LD      Y141  ; ﾚｰﾝ7上段(中間)ﾜｰｸｽﾄｯﾊﾟｰ開
      ANI     X6B  ; ﾚｰﾝ7上段(中間)ﾜｰｸｽﾄｯﾊﾟｰ開端
      ORB
      LD      T49  ; ﾚｰﾝ7上段(中間)ﾜｰｸｽﾄｯﾊﾟｰ動作異常
      ANI     M20  ; 異常ﾘｾｯﾄ
      ORB
      OUT     T49 K70  ; ﾚｰﾝ7上段(中間)ﾜｰｸｽﾄｯﾊﾟｰ動作異常
574   LD      X6C  ; ﾚｰﾝ7上段(中間)切出し上昇端
      AND     X6D  ; ﾚｰﾝ7上段(中間)切出し下降端
      LD      M56  ; ﾚｰﾝ7上段(中間)切出しLS異常
      ANI     M20  ; 異常ﾘｾｯﾄ
      ORB
      OUT     M56  ; ﾚｰﾝ7上段(中間)切出しLS異常
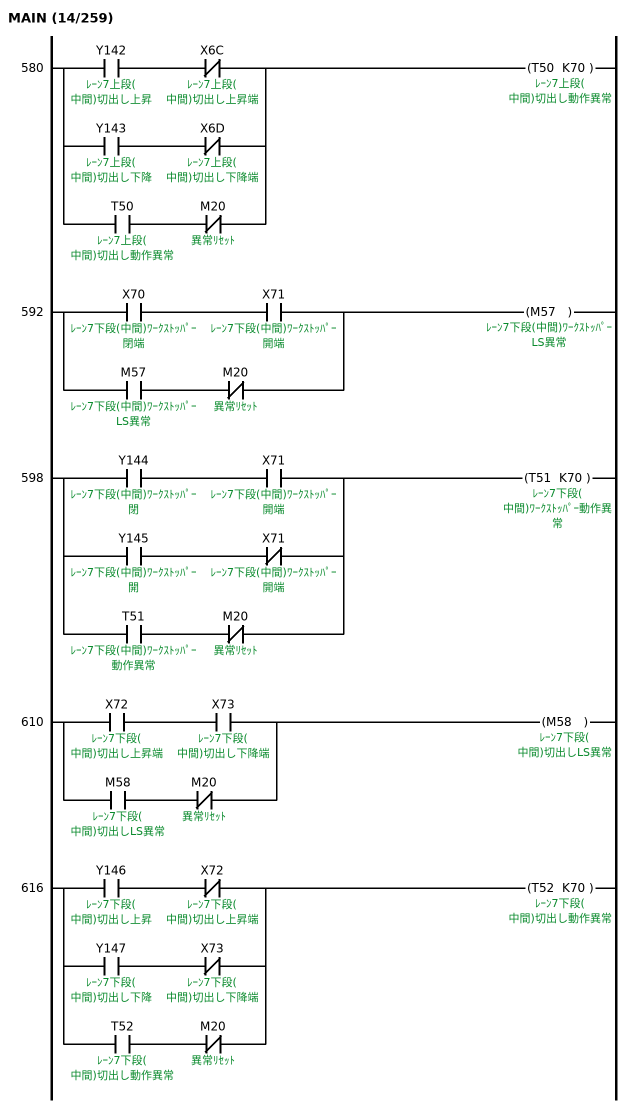
580   LD      Y142  ; ﾚｰﾝ7上段(中間)切出し上昇
      ANI     X6C  ; ﾚｰﾝ7上段(中間)切出し上昇端
      LD      Y143  ; ﾚｰﾝ7上段(中間)切出し下降
      ANI     X6D  ; ﾚｰﾝ7上段(中間)切出し下降端
      ORB
      LD      T50  ; ﾚｰﾝ7上段(中間)切出し動作異常
      ANI     M20  ; 異常ﾘｾｯﾄ
      ORB
      OUT     T50 K70  ; ﾚｰﾝ7上段(中間)切出し動作異常
592   LD      X70  ; ﾚｰﾝ7下段(中間)ﾜｰｸｽﾄｯﾊﾟｰ閉端
      AND     X71  ; ﾚｰﾝ7下段(中間)ﾜｰｸｽﾄｯﾊﾟｰ開端
      LD      M57  ; ﾚｰﾝ7下段(中間)ﾜｰｸｽﾄｯﾊﾟｰLS異常
      ANI     M20  ; 異常ﾘｾｯﾄ
      ORB
      OUT     M57  ; ﾚｰﾝ7下段(中間)ﾜｰｸｽﾄｯﾊﾟｰLS異常
598   LD      Y144  ; ﾚｰﾝ7下段(中間)ﾜｰｸｽﾄｯﾊﾟｰ閉
      AND     X71  ; ﾚｰﾝ7下段(中間)ﾜｰｸｽﾄｯﾊﾟｰ開端
      LD      Y145  ; ﾚｰﾝ7下段(中間)ﾜｰｸｽﾄｯﾊﾟｰ開
      ANI     X71  ; ﾚｰﾝ7下段(中間)ﾜｰｸｽﾄｯﾊﾟｰ開端
      ORB
      LD      T51  ; ﾚｰﾝ7下段(中間)ﾜｰｸｽﾄｯﾊﾟｰ動作異常
      ANI     M20  ; 異常ﾘｾｯﾄ
      ORB
      OUT     T51 K70  ; ﾚｰﾝ7下段(中間)ﾜｰｸｽﾄｯﾊﾟｰ動作異常
610   LD      X72  ; ﾚｰﾝ7下段(中間)切出し上昇端
      AND     X73  ; ﾚｰﾝ7下段(中間)切出し下降端
      LD      M58  ; ﾚｰﾝ7下段(中間)切出しLS異常
      ANI     M20  ; 異常ﾘｾｯﾄ
      ORB
      OUT     M58  ; ﾚｰﾝ7下段(中間)切出しLS異常
616   LD      Y146  ; ﾚｰﾝ7下段(中間)切出し上昇
      ANI     X72  ; ﾚｰﾝ7下段(中間)切出し上昇端
      LD      Y147  ; ﾚｰﾝ7下段(中間)切出し下降
      ANI     X73  ; ﾚｰﾝ7下段(中間)切出し下降端
      ORB
      LD      T52  ; ﾚｰﾝ7下段(中間)切出し動作異常
      ANI     M20  ; 異常ﾘｾｯﾄ
      ORB
      OUT     T52 K70  ; ﾚｰﾝ7下段(中間)切出し動作異常
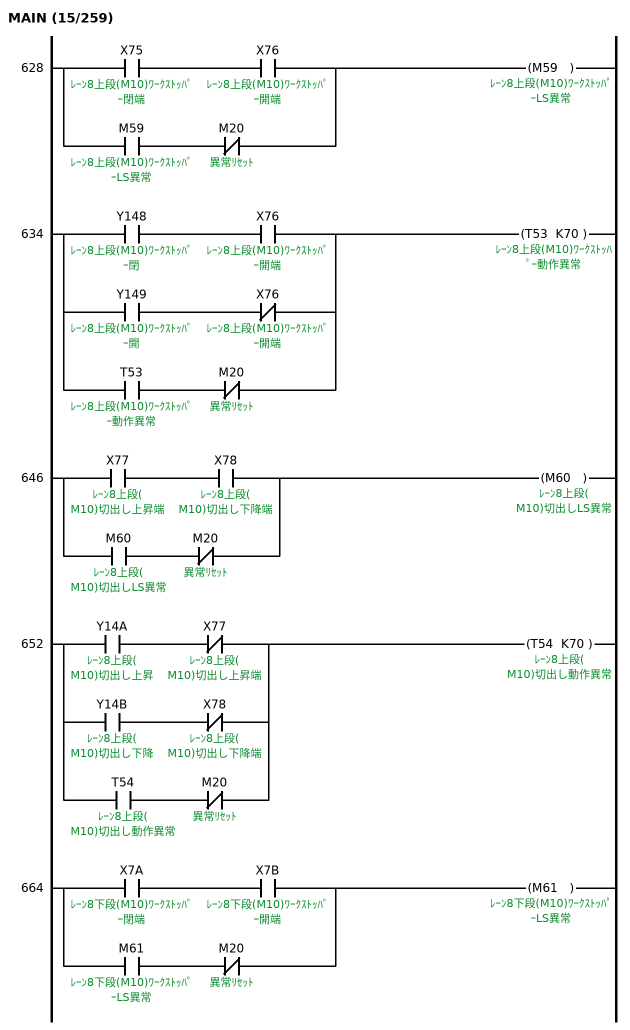
628   LD      X75  ; ﾚｰﾝ8上段(M10)ﾜｰｸｽﾄｯﾊﾟｰ閉端
      AND     X76  ; ﾚｰﾝ8上段(M10)ﾜｰｸｽﾄｯﾊﾟｰ開端
      LD      M59  ; ﾚｰﾝ8上段(M10)ﾜｰｸｽﾄｯﾊﾟｰLS異常
      ANI     M20  ; 異常ﾘｾｯﾄ
      ORB
      OUT     M59  ; ﾚｰﾝ8上段(M10)ﾜｰｸｽﾄｯﾊﾟｰLS異常
634   LD      Y148  ; ﾚｰﾝ8上段(M10)ﾜｰｸｽﾄｯﾊﾟｰ閉
      AND     X76  ; ﾚｰﾝ8上段(M10)ﾜｰｸｽﾄｯﾊﾟｰ開端
      LD      Y149  ; ﾚｰﾝ8上段(M10)ﾜｰｸｽﾄｯﾊﾟｰ開
      ANI     X76  ; ﾚｰﾝ8上段(M10)ﾜｰｸｽﾄｯﾊﾟｰ開端
      ORB
      LD      T53  ; ﾚｰﾝ8上段(M10)ﾜｰｸｽﾄｯﾊﾟｰ動作異常
      ANI     M20  ; 異常ﾘｾｯﾄ
      ORB
      OUT     T53 K70  ; ﾚｰﾝ8上段(M10)ﾜｰｸｽﾄｯﾊﾟｰ動作異常
646   LD      X77  ; ﾚｰﾝ8上段(M10)切出し上昇端
      AND     X78  ; ﾚｰﾝ8上段(M10)切出し下降端
      LD      M60  ; ﾚｰﾝ8上段(M10)切出しLS異常
      ANI     M20  ; 異常ﾘｾｯﾄ
      ORB
      OUT     M60  ; ﾚｰﾝ8上段(M10)切出しLS異常
652   LD      Y14A  ; ﾚｰﾝ8上段(M10)切出し上昇
      ANI     X77  ; ﾚｰﾝ8上段(M10)切出し上昇端
      LD      Y14B  ; ﾚｰﾝ8上段(M10)切出し下降
      ANI     X78  ; ﾚｰﾝ8上段(M10)切出し下降端
      ORB
      LD      T54  ; ﾚｰﾝ8上段(M10)切出し動作異常
      ANI     M20  ; 異常ﾘｾｯﾄ
      ORB
      OUT     T54 K70  ; ﾚｰﾝ8上段(M10)切出し動作異常
664   LD      X7A  ; ﾚｰﾝ8下段(M10)ﾜｰｸｽﾄｯﾊﾟｰ閉端
      AND     X7B  ; ﾚｰﾝ8下段(M10)ﾜｰｸｽﾄｯﾊﾟｰ開端
      LD      M61  ; ﾚｰﾝ8下段(M10)ﾜｰｸｽﾄｯﾊﾟｰLS異常
      ANI     M20  ; 異常ﾘｾｯﾄ
      ORB
      OUT     M61  ; ﾚｰﾝ8下段(M10)ﾜｰｸｽﾄｯﾊﾟｰLS異常
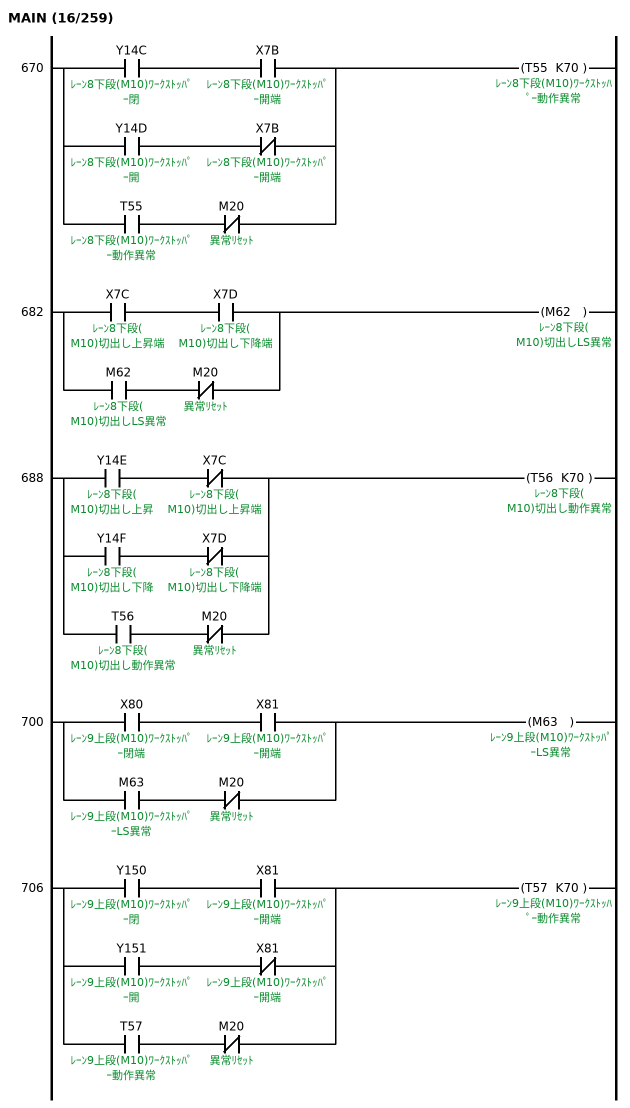
670   LD      Y14C  ; ﾚｰﾝ8下段(M10)ﾜｰｸｽﾄｯﾊﾟｰ閉
      AND     X7B  ; ﾚｰﾝ8下段(M10)ﾜｰｸｽﾄｯﾊﾟｰ開端
      LD      Y14D  ; ﾚｰﾝ8下段(M10)ﾜｰｸｽﾄｯﾊﾟｰ開
      ANI     X7B  ; ﾚｰﾝ8下段(M10)ﾜｰｸｽﾄｯﾊﾟｰ開端
      ORB
      LD      T55  ; ﾚｰﾝ8下段(M10)ﾜｰｸｽﾄｯﾊﾟｰ動作異常
      ANI     M20  ; 異常ﾘｾｯﾄ
      ORB
      OUT     T55 K70  ; ﾚｰﾝ8下段(M10)ﾜｰｸｽﾄｯﾊﾟｰ動作異常
682   LD      X7C  ; ﾚｰﾝ8下段(M10)切出し上昇端
      AND     X7D  ; ﾚｰﾝ8下段(M10)切出し下降端
      LD      M62  ; ﾚｰﾝ8下段(M10)切出しLS異常
      ANI     M20  ; 異常ﾘｾｯﾄ
      ORB
      OUT     M62  ; ﾚｰﾝ8下段(M10)切出しLS異常
688   LD      Y14E  ; ﾚｰﾝ8下段(M10)切出し上昇
      ANI     X7C  ; ﾚｰﾝ8下段(M10)切出し上昇端
      LD      Y14F  ; ﾚｰﾝ8下段(M10)切出し下降
      ANI     X7D  ; ﾚｰﾝ8下段(M10)切出し下降端
      ORB
      LD      T56  ; ﾚｰﾝ8下段(M10)切出し動作異常
      ANI     M20  ; 異常ﾘｾｯﾄ
      ORB
      OUT     T56 K70  ; ﾚｰﾝ8下段(M10)切出し動作異常
700   LD      X80  ; ﾚｰﾝ9上段(M10)ﾜｰｸｽﾄｯﾊﾟｰ閉端
      AND     X81  ; ﾚｰﾝ9上段(M10)ﾜｰｸｽﾄｯﾊﾟｰ開端
      LD      M63  ; ﾚｰﾝ9上段(M10)ﾜｰｸｽﾄｯﾊﾟｰLS異常
      ANI     M20  ; 異常ﾘｾｯﾄ
      ORB
      OUT     M63  ; ﾚｰﾝ9上段(M10)ﾜｰｸｽﾄｯﾊﾟｰLS異常
706   LD      Y150  ; ﾚｰﾝ9上段(M10)ﾜｰｸｽﾄｯﾊﾟｰ閉
      AND     X81  ; ﾚｰﾝ9上段(M10)ﾜｰｸｽﾄｯﾊﾟｰ開端
      LD      Y151  ; ﾚｰﾝ9上段(M10)ﾜｰｸｽﾄｯﾊﾟｰ開
      ANI     X81  ; ﾚｰﾝ9上段(M10)ﾜｰｸｽﾄｯﾊﾟｰ開端
      ORB
      LD      T57  ; ﾚｰﾝ9上段(M10)ﾜｰｸｽﾄｯﾊﾟｰ動作異常
      ANI     M20  ; 異常ﾘｾｯﾄ
      ORB
      OUT     T57 K70  ; ﾚｰﾝ9上段(M10)ﾜｰｸｽﾄｯﾊﾟｰ動作異常
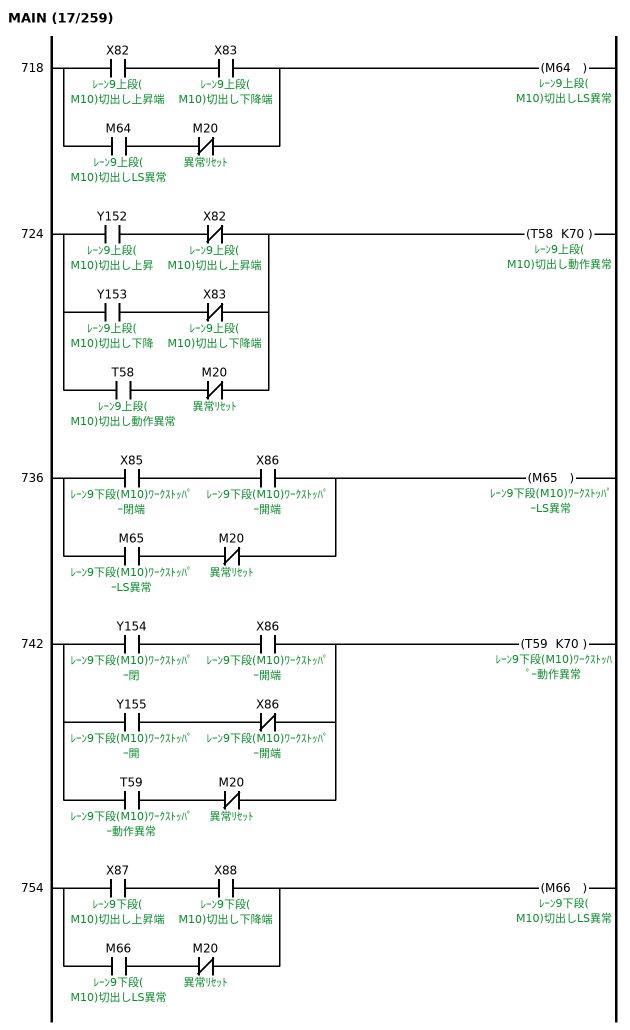
718   LD      X82  ; ﾚｰﾝ9上段(M10)切出し上昇端
      AND     X83  ; ﾚｰﾝ9上段(M10)切出し下降端
      LD      M64  ; ﾚｰﾝ9上段(M10)切出しLS異常
      ANI     M20  ; 異常ﾘｾｯﾄ
      ORB
      OUT     M64  ; ﾚｰﾝ9上段(M10)切出しLS異常
724   LD      Y152  ; ﾚｰﾝ9上段(M10)切出し上昇
      ANI     X82  ; ﾚｰﾝ9上段(M10)切出し上昇端
      LD      Y153  ; ﾚｰﾝ9上段(M10)切出し下降
      ANI     X83  ; ﾚｰﾝ9上段(M10)切出し下降端
      ORB
      LD      T58  ; ﾚｰﾝ9上段(M10)切出し動作異常
      ANI     M20  ; 異常ﾘｾｯﾄ
      ORB
      OUT     T58 K70  ; ﾚｰﾝ9上段(M10)切出し動作異常
736   LD      X85  ; ﾚｰﾝ9下段(M10)ﾜｰｸｽﾄｯﾊﾟｰ閉端
      AND     X86  ; ﾚｰﾝ9下段(M10)ﾜｰｸｽﾄｯﾊﾟｰ開端
      LD      M65  ; ﾚｰﾝ9下段(M10)ﾜｰｸｽﾄｯﾊﾟｰLS異常
      ANI     M20  ; 異常ﾘｾｯﾄ
      ORB
      OUT     M65  ; ﾚｰﾝ9下段(M10)ﾜｰｸｽﾄｯﾊﾟｰLS異常
742   LD      Y154  ; ﾚｰﾝ9下段(M10)ﾜｰｸｽﾄｯﾊﾟｰ閉
      AND     X86  ; ﾚｰﾝ9下段(M10)ﾜｰｸｽﾄｯﾊﾟｰ開端
      LD      Y155  ; ﾚｰﾝ9下段(M10)ﾜｰｸｽﾄｯﾊﾟｰ開
      ANI     X86  ; ﾚｰﾝ9下段(M10)ﾜｰｸｽﾄｯﾊﾟｰ開端
      ORB
      LD      T59  ; ﾚｰﾝ9下段(M10)ﾜｰｸｽﾄｯﾊﾟｰ動作異常
      ANI     M20  ; 異常ﾘｾｯﾄ
      ORB
      OUT     T59 K70  ; ﾚｰﾝ9下段(M10)ﾜｰｸｽﾄｯﾊﾟｰ動作異常
754   LD      X87  ; ﾚｰﾝ9下段(M10)切出し上昇端
      AND     X88  ; ﾚｰﾝ9下段(M10)切出し下降端
      LD      M66  ; ﾚｰﾝ9下段(M10)切出しLS異常
      ANI     M20  ; 異常ﾘｾｯﾄ
      ORB
      OUT     M66  ; ﾚｰﾝ9下段(M10)切出しLS異常
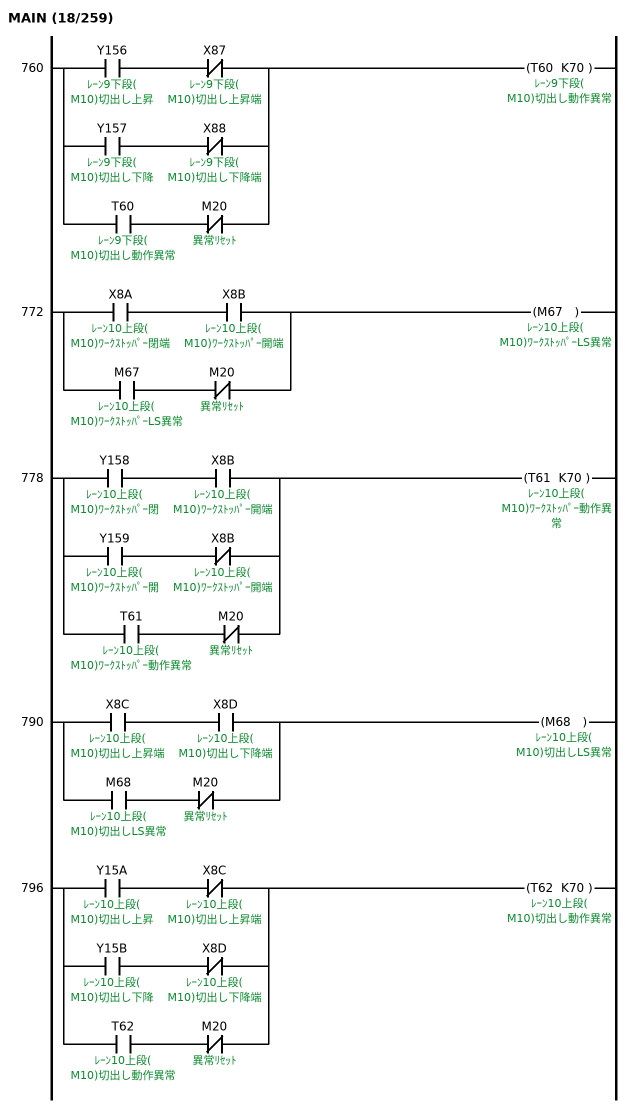
760   LD      Y156  ; ﾚｰﾝ9下段(M10)切出し上昇
      ANI     X87  ; ﾚｰﾝ9下段(M10)切出し上昇端
      LD      Y157  ; ﾚｰﾝ9下段(M10)切出し下降
      ANI     X88  ; ﾚｰﾝ9下段(M10)切出し下降端
      ORB
      LD      T60  ; ﾚｰﾝ9下段(M10)切出し動作異常
      ANI     M20  ; 異常ﾘｾｯﾄ
      ORB
      OUT     T60 K70  ; ﾚｰﾝ9下段(M10)切出し動作異常
772   LD      X8A  ; ﾚｰﾝ10上段(M10)ﾜｰｸｽﾄｯﾊﾟｰ閉端
      AND     X8B  ; ﾚｰﾝ10上段(M10)ﾜｰｸｽﾄｯﾊﾟｰ開端
      LD      M67  ; ﾚｰﾝ10上段(M10)ﾜｰｸｽﾄｯﾊﾟｰLS異常
      ANI     M20  ; 異常ﾘｾｯﾄ
      ORB
      OUT     M67  ; ﾚｰﾝ10上段(M10)ﾜｰｸｽﾄｯﾊﾟｰLS異常
778   LD      Y158  ; ﾚｰﾝ10上段(M10)ﾜｰｸｽﾄｯﾊﾟｰ閉
      AND     X8B  ; ﾚｰﾝ10上段(M10)ﾜｰｸｽﾄｯﾊﾟｰ開端
      LD      Y159  ; ﾚｰﾝ10上段(M10)ﾜｰｸｽﾄｯﾊﾟｰ開
      ANI     X8B  ; ﾚｰﾝ10上段(M10)ﾜｰｸｽﾄｯﾊﾟｰ開端
      ORB
      LD      T61  ; ﾚｰﾝ10上段(M10)ﾜｰｸｽﾄｯﾊﾟｰ動作異常
      ANI     M20  ; 異常ﾘｾｯﾄ
      ORB
      OUT     T61 K70  ; ﾚｰﾝ10上段(M10)ﾜｰｸｽﾄｯﾊﾟｰ動作異常
790   LD      X8C  ; ﾚｰﾝ10上段(M10)切出し上昇端
      AND     X8D  ; ﾚｰﾝ10上段(M10)切出し下降端
      LD      M68  ; ﾚｰﾝ10上段(M10)切出しLS異常
      ANI     M20  ; 異常ﾘｾｯﾄ
      ORB
      OUT     M68  ; ﾚｰﾝ10上段(M10)切出しLS異常
796   LD      Y15A  ; ﾚｰﾝ10上段(M10)切出し上昇
      ANI     X8C  ; ﾚｰﾝ10上段(M10)切出し上昇端
      LD      Y15B  ; ﾚｰﾝ10上段(M10)切出し下降
      ANI     X8D  ; ﾚｰﾝ10上段(M10)切出し下降端
      ORB
      LD      T62  ; ﾚｰﾝ10上段(M10)切出し動作異常
      ANI     M20  ; 異常ﾘｾｯﾄ
      ORB
      OUT     T62 K70  ; ﾚｰﾝ10上段(M10)切出し動作異常
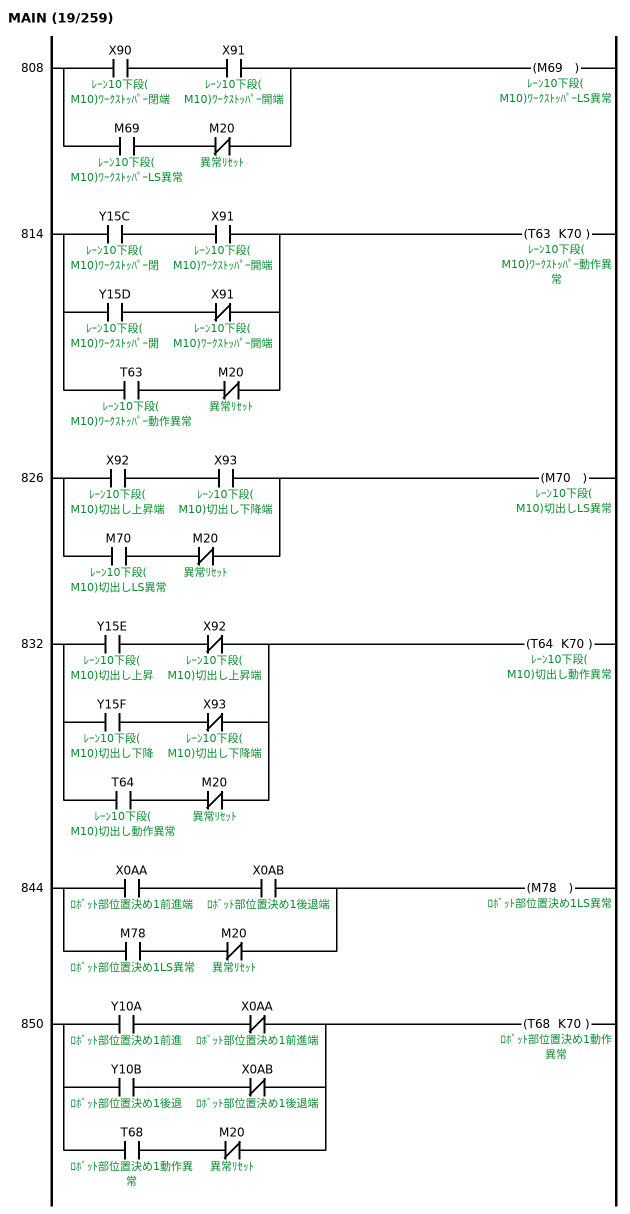
808   LD      X90  ; ﾚｰﾝ10下段(M10)ﾜｰｸｽﾄｯﾊﾟｰ閉端
      AND     X91  ; ﾚｰﾝ10下段(M10)ﾜｰｸｽﾄｯﾊﾟｰ開端
      LD      M69  ; ﾚｰﾝ10下段(M10)ﾜｰｸｽﾄｯﾊﾟｰLS異常
      ANI     M20  ; 異常ﾘｾｯﾄ
      ORB
      OUT     M69  ; ﾚｰﾝ10下段(M10)ﾜｰｸｽﾄｯﾊﾟｰLS異常
814   LD      Y15C  ; ﾚｰﾝ10下段(M10)ﾜｰｸｽﾄｯﾊﾟｰ閉
      AND     X91  ; ﾚｰﾝ10下段(M10)ﾜｰｸｽﾄｯﾊﾟｰ開端
      LD      Y15D  ; ﾚｰﾝ10下段(M10)ﾜｰｸｽﾄｯﾊﾟｰ開
      ANI     X91  ; ﾚｰﾝ10下段(M10)ﾜｰｸｽﾄｯﾊﾟｰ開端
      ORB
      LD      T63  ; ﾚｰﾝ10下段(M10)ﾜｰｸｽﾄｯﾊﾟｰ動作異常
      ANI     M20  ; 異常ﾘｾｯﾄ
      ORB
      OUT     T63 K70  ; ﾚｰﾝ10下段(M10)ﾜｰｸｽﾄｯﾊﾟｰ動作異常
826   LD      X92  ; ﾚｰﾝ10下段(M10)切出し上昇端
      AND     X93  ; ﾚｰﾝ10下段(M10)切出し下降端
      LD      M70  ; ﾚｰﾝ10下段(M10)切出しLS異常
      ANI     M20  ; 異常ﾘｾｯﾄ
      ORB
      OUT     M70  ; ﾚｰﾝ10下段(M10)切出しLS異常
832   LD      Y15E  ; ﾚｰﾝ10下段(M10)切出し上昇
      ANI     X92  ; ﾚｰﾝ10下段(M10)切出し上昇端
      LD      Y15F  ; ﾚｰﾝ10下段(M10)切出し下降
      ANI     X93  ; ﾚｰﾝ10下段(M10)切出し下降端
      ORB
      LD      T64  ; ﾚｰﾝ10下段(M10)切出し動作異常
      ANI     M20  ; 異常ﾘｾｯﾄ
      ORB
      OUT     T64 K70  ; ﾚｰﾝ10下段(M10)切出し動作異常
844   LD      X0AA  ; ﾛﾎﾞｯﾄ部位置決め1前進端
      AND     X0AB  ; ﾛﾎﾞｯﾄ部位置決め1後退端
      LD      M78  ; ﾛﾎﾞｯﾄ部位置決め1LS異常
      ANI     M20  ; 異常ﾘｾｯﾄ
      ORB
      OUT     M78  ; ﾛﾎﾞｯﾄ部位置決め1LS異常
850   LD      Y10A  ; ﾛﾎﾞｯﾄ部位置決め1前進
      ANI     X0AA  ; ﾛﾎﾞｯﾄ部位置決め1前進端
      LD      Y10B  ; ﾛﾎﾞｯﾄ部位置決め1後退
      ANI     X0AB  ; ﾛﾎﾞｯﾄ部位置決め1後退端
      ORB
      LD      T68  ; ﾛﾎﾞｯﾄ部位置決め1動作異常
      ANI     M20  ; 異常ﾘｾｯﾄ
      ORB
      OUT     T68 K70  ; ﾛﾎﾞｯﾄ部位置決め1動作異常
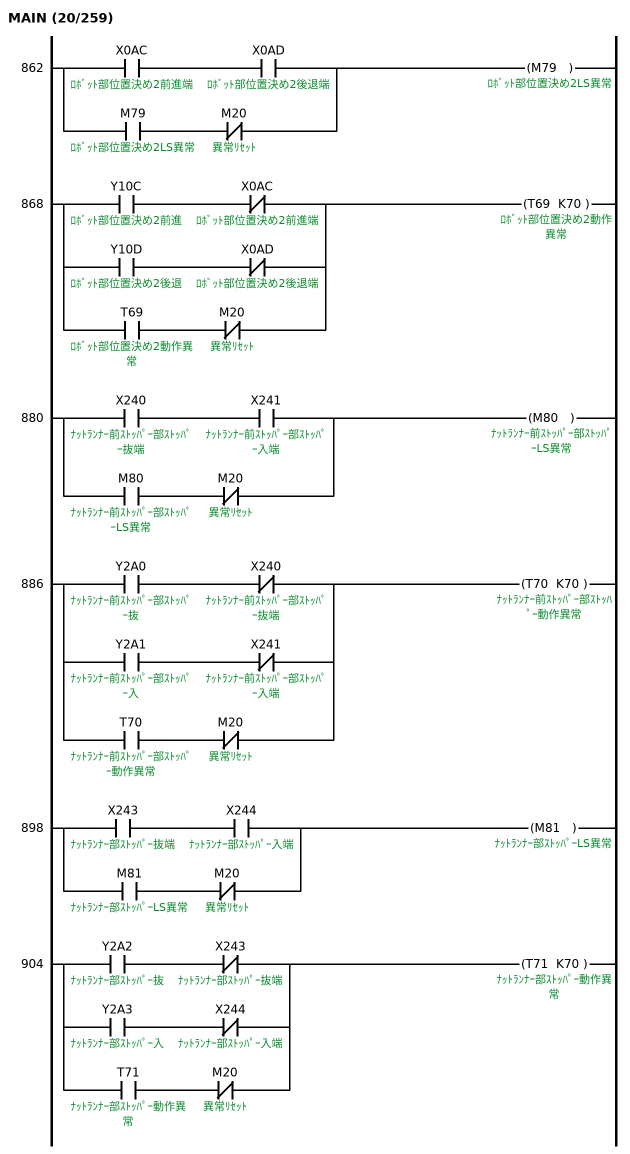
862   LD      X0AC  ; ﾛﾎﾞｯﾄ部位置決め2前進端
      AND     X0AD  ; ﾛﾎﾞｯﾄ部位置決め2後退端
      LD      M79  ; ﾛﾎﾞｯﾄ部位置決め2LS異常
      ANI     M20  ; 異常ﾘｾｯﾄ
      ORB
      OUT     M79  ; ﾛﾎﾞｯﾄ部位置決め2LS異常
868   LD      Y10C  ; ﾛﾎﾞｯﾄ部位置決め2前進
      ANI     X0AC  ; ﾛﾎﾞｯﾄ部位置決め2前進端
      LD      Y10D  ; ﾛﾎﾞｯﾄ部位置決め2後退
      ANI     X0AD  ; ﾛﾎﾞｯﾄ部位置決め2後退端
      ORB
      LD      T69  ; ﾛﾎﾞｯﾄ部位置決め2動作異常
      ANI     M20  ; 異常ﾘｾｯﾄ
      ORB
      OUT     T69 K70  ; ﾛﾎﾞｯﾄ部位置決め2動作異常
880   LD      X240  ; ﾅｯﾄﾗﾝﾅｰ前ｽﾄｯﾊﾟｰ部ｽﾄｯﾊﾟｰ抜端
      AND     X241  ; ﾅｯﾄﾗﾝﾅｰ前ｽﾄｯﾊﾟｰ部ｽﾄｯﾊﾟｰ入端
      LD      M80  ; ﾅｯﾄﾗﾝﾅｰ前ｽﾄｯﾊﾟｰ部ｽﾄｯﾊﾟｰLS異常
      ANI     M20  ; 異常ﾘｾｯﾄ
      ORB
      OUT     M80  ; ﾅｯﾄﾗﾝﾅｰ前ｽﾄｯﾊﾟｰ部ｽﾄｯﾊﾟｰLS異常
886   LD      Y2A0  ; ﾅｯﾄﾗﾝﾅｰ前ｽﾄｯﾊﾟｰ部ｽﾄｯﾊﾟｰ抜
      ANI     X240  ; ﾅｯﾄﾗﾝﾅｰ前ｽﾄｯﾊﾟｰ部ｽﾄｯﾊﾟｰ抜端
      LD      Y2A1  ; ﾅｯﾄﾗﾝﾅｰ前ｽﾄｯﾊﾟｰ部ｽﾄｯﾊﾟｰ入
      ANI     X241  ; ﾅｯﾄﾗﾝﾅｰ前ｽﾄｯﾊﾟｰ部ｽﾄｯﾊﾟｰ入端
      ORB
      LD      T70  ; ﾅｯﾄﾗﾝﾅｰ前ｽﾄｯﾊﾟｰ部ｽﾄｯﾊﾟｰ動作異常
      ANI     M20  ; 異常ﾘｾｯﾄ
      ORB
      OUT     T70 K70  ; ﾅｯﾄﾗﾝﾅｰ前ｽﾄｯﾊﾟｰ部ｽﾄｯﾊﾟｰ動作異常
898   LD      X243  ; ﾅｯﾄﾗﾝﾅｰ部ｽﾄｯﾊﾟｰ抜端
      AND     X244  ; ﾅｯﾄﾗﾝﾅｰ部ｽﾄｯﾊﾟｰ入端
      LD      M81  ; ﾅｯﾄﾗﾝﾅｰ部ｽﾄｯﾊﾟｰLS異常
      ANI     M20  ; 異常ﾘｾｯﾄ
      ORB
      OUT     M81  ; ﾅｯﾄﾗﾝﾅｰ部ｽﾄｯﾊﾟｰLS異常
904   LD      Y2A2  ; ﾅｯﾄﾗﾝﾅｰ部ｽﾄｯﾊﾟｰ抜
      ANI     X243  ; ﾅｯﾄﾗﾝﾅｰ部ｽﾄｯﾊﾟｰ抜端
      LD      Y2A3  ; ﾅｯﾄﾗﾝﾅｰ部ｽﾄｯﾊﾟｰ入
      ANI     X244  ; ﾅｯﾄﾗﾝﾅｰ部ｽﾄｯﾊﾟｰ入端
      ORB
      LD      T71  ; ﾅｯﾄﾗﾝﾅｰ部ｽﾄｯﾊﾟｰ動作異常
      ANI     M20  ; 異常ﾘｾｯﾄ
      ORB
      OUT     T71 K70  ; ﾅｯﾄﾗﾝﾅｰ部ｽﾄｯﾊﾟｰ動作異常
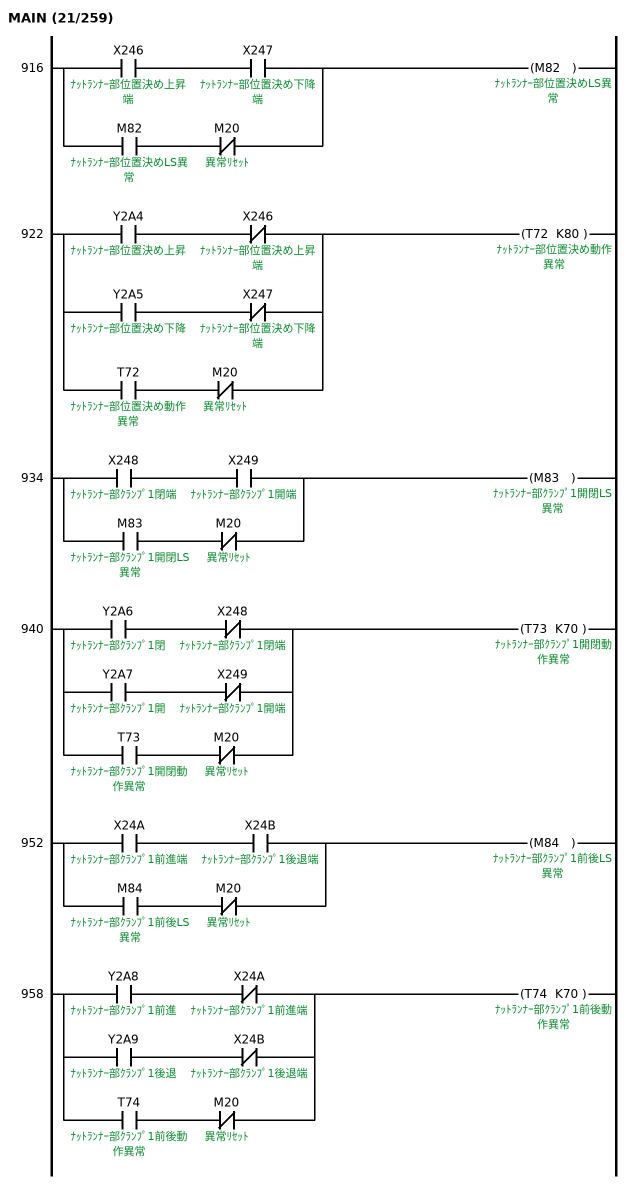
916   LD      X246  ; ﾅｯﾄﾗﾝﾅｰ部位置決め上昇端
      AND     X247  ; ﾅｯﾄﾗﾝﾅｰ部位置決め下降端
      LD      M82  ; ﾅｯﾄﾗﾝﾅｰ部位置決めLS異常
      ANI     M20  ; 異常ﾘｾｯﾄ
      ORB
      OUT     M82  ; ﾅｯﾄﾗﾝﾅｰ部位置決めLS異常
922   LD      Y2A4  ; ﾅｯﾄﾗﾝﾅｰ部位置決め上昇
      ANI     X246  ; ﾅｯﾄﾗﾝﾅｰ部位置決め上昇端
      LD      Y2A5  ; ﾅｯﾄﾗﾝﾅｰ部位置決め下降
      ANI     X247  ; ﾅｯﾄﾗﾝﾅｰ部位置決め下降端
      ORB
      LD      T72  ; ﾅｯﾄﾗﾝﾅｰ部位置決め動作異常
      ANI     M20  ; 異常ﾘｾｯﾄ
      ORB
      OUT     T72 K80  ; ﾅｯﾄﾗﾝﾅｰ部位置決め動作異常
934   LD      X248  ; ﾅｯﾄﾗﾝﾅｰ部ｸﾗﾝﾌﾟ1閉端
      AND     X249  ; ﾅｯﾄﾗﾝﾅｰ部ｸﾗﾝﾌﾟ1開端
      LD      M83  ; ﾅｯﾄﾗﾝﾅｰ部ｸﾗﾝﾌﾟ1開閉LS異常
      ANI     M20  ; 異常ﾘｾｯﾄ
      ORB
      OUT     M83  ; ﾅｯﾄﾗﾝﾅｰ部ｸﾗﾝﾌﾟ1開閉LS異常
940   LD      Y2A6  ; ﾅｯﾄﾗﾝﾅｰ部ｸﾗﾝﾌﾟ1閉
      ANI     X248  ; ﾅｯﾄﾗﾝﾅｰ部ｸﾗﾝﾌﾟ1閉端
      LD      Y2A7  ; ﾅｯﾄﾗﾝﾅｰ部ｸﾗﾝﾌﾟ1開
      ANI     X249  ; ﾅｯﾄﾗﾝﾅｰ部ｸﾗﾝﾌﾟ1開端
      ORB
      LD      T73  ; ﾅｯﾄﾗﾝﾅｰ部ｸﾗﾝﾌﾟ1開閉動作異常
      ANI     M20  ; 異常ﾘｾｯﾄ
      ORB
      OUT     T73 K70  ; ﾅｯﾄﾗﾝﾅｰ部ｸﾗﾝﾌﾟ1開閉動作異常
952   LD      X24A  ; ﾅｯﾄﾗﾝﾅｰ部ｸﾗﾝﾌﾟ1前進端
      AND     X24B  ; ﾅｯﾄﾗﾝﾅｰ部ｸﾗﾝﾌﾟ1後退端
      LD      M84  ; ﾅｯﾄﾗﾝﾅｰ部ｸﾗﾝﾌﾟ1前後LS異常
      ANI     M20  ; 異常ﾘｾｯﾄ
      ORB
      OUT     M84  ; ﾅｯﾄﾗﾝﾅｰ部ｸﾗﾝﾌﾟ1前後LS異常
958   LD      Y2A8  ; ﾅｯﾄﾗﾝﾅｰ部ｸﾗﾝﾌﾟ1前進
      ANI     X24A  ; ﾅｯﾄﾗﾝﾅｰ部ｸﾗﾝﾌﾟ1前進端
      LD      Y2A9  ; ﾅｯﾄﾗﾝﾅｰ部ｸﾗﾝﾌﾟ1後退
      ANI     X24B  ; ﾅｯﾄﾗﾝﾅｰ部ｸﾗﾝﾌﾟ1後退端
      ORB
      LD      T74  ; ﾅｯﾄﾗﾝﾅｰ部ｸﾗﾝﾌﾟ1前後動作異常
      ANI     M20  ; 異常ﾘｾｯﾄ
      ORB
      OUT     T74 K70  ; ﾅｯﾄﾗﾝﾅｰ部ｸﾗﾝﾌﾟ1前後動作異常
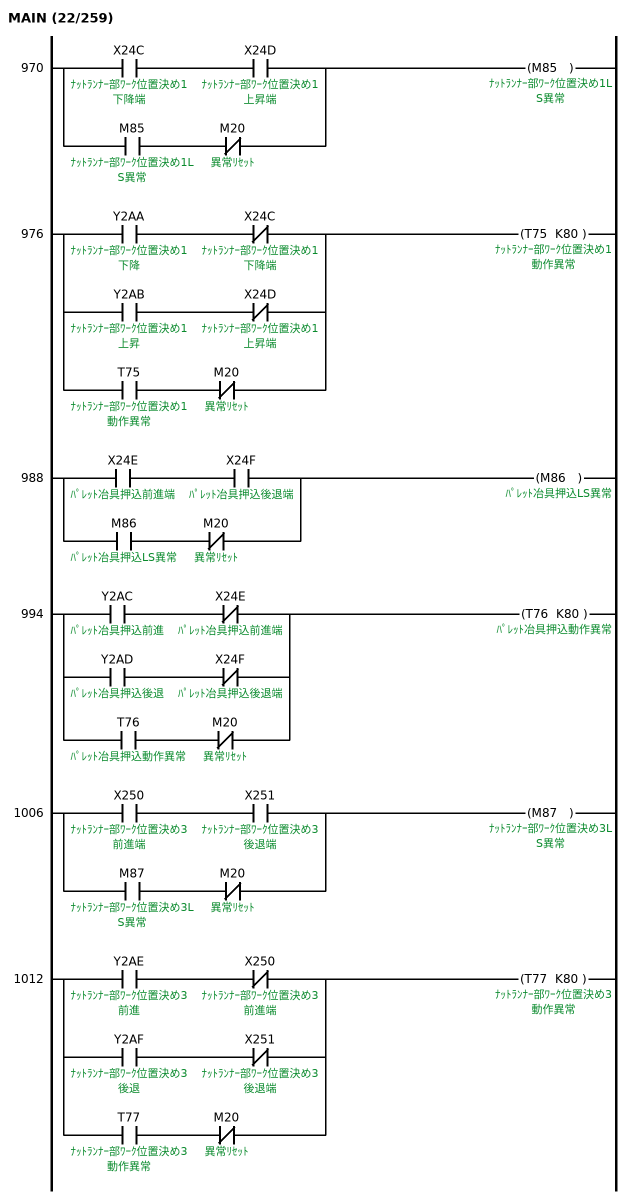
970   LD      X24C  ; ﾅｯﾄﾗﾝﾅｰ部ﾜｰｸ位置決め1下降端
      AND     X24D  ; ﾅｯﾄﾗﾝﾅｰ部ﾜｰｸ位置決め1上昇端
      LD      M85  ; ﾅｯﾄﾗﾝﾅｰ部ﾜｰｸ位置決め1LS異常
      ANI     M20  ; 異常ﾘｾｯﾄ
      ORB
      OUT     M85  ; ﾅｯﾄﾗﾝﾅｰ部ﾜｰｸ位置決め1LS異常
976   LD      Y2AA  ; ﾅｯﾄﾗﾝﾅｰ部ﾜｰｸ位置決め1下降
      ANI     X24C  ; ﾅｯﾄﾗﾝﾅｰ部ﾜｰｸ位置決め1下降端
      LD      Y2AB  ; ﾅｯﾄﾗﾝﾅｰ部ﾜｰｸ位置決め1上昇
      ANI     X24D  ; ﾅｯﾄﾗﾝﾅｰ部ﾜｰｸ位置決め1上昇端
      ORB
      LD      T75  ; ﾅｯﾄﾗﾝﾅｰ部ﾜｰｸ位置決め1動作異常
      ANI     M20  ; 異常ﾘｾｯﾄ
      ORB
      OUT     T75 K80  ; ﾅｯﾄﾗﾝﾅｰ部ﾜｰｸ位置決め1動作異常
988   LD      X24E  ; ﾊﾟﾚｯﾄ冶具押込前進端
      AND     X24F  ; ﾊﾟﾚｯﾄ冶具押込後退端
      LD      M86  ; ﾊﾟﾚｯﾄ冶具押込LS異常
      ANI     M20  ; 異常ﾘｾｯﾄ
      ORB
      OUT     M86  ; ﾊﾟﾚｯﾄ冶具押込LS異常
994   LD      Y2AC  ; ﾊﾟﾚｯﾄ冶具押込前進
      ANI     X24E  ; ﾊﾟﾚｯﾄ冶具押込前進端
      LD      Y2AD  ; ﾊﾟﾚｯﾄ冶具押込後退
      ANI     X24F  ; ﾊﾟﾚｯﾄ冶具押込後退端
      ORB
      LD      T76  ; ﾊﾟﾚｯﾄ冶具押込動作異常
      ANI     M20  ; 異常ﾘｾｯﾄ
      ORB
      OUT     T76 K80  ; ﾊﾟﾚｯﾄ冶具押込動作異常
1006  LD      X250  ; ﾅｯﾄﾗﾝﾅｰ部ﾜｰｸ位置決め3前進端
      AND     X251  ; ﾅｯﾄﾗﾝﾅｰ部ﾜｰｸ位置決め3後退端
      LD      M87  ; ﾅｯﾄﾗﾝﾅｰ部ﾜｰｸ位置決め3LS異常
      ANI     M20  ; 異常ﾘｾｯﾄ
      ORB
      OUT     M87  ; ﾅｯﾄﾗﾝﾅｰ部ﾜｰｸ位置決め3LS異常
1012  LD      Y2AE  ; ﾅｯﾄﾗﾝﾅｰ部ﾜｰｸ位置決め3前進
      ANI     X250  ; ﾅｯﾄﾗﾝﾅｰ部ﾜｰｸ位置決め3前進端
      LD      Y2AF  ; ﾅｯﾄﾗﾝﾅｰ部ﾜｰｸ位置決め3後退
      ANI     X251  ; ﾅｯﾄﾗﾝﾅｰ部ﾜｰｸ位置決め3後退端
      ORB
      LD      T77  ; ﾅｯﾄﾗﾝﾅｰ部ﾜｰｸ位置決め3動作異常
      ANI     M20  ; 異常ﾘｾｯﾄ
      ORB
      OUT     T77 K80  ; ﾅｯﾄﾗﾝﾅｰ部ﾜｰｸ位置決め3動作異常
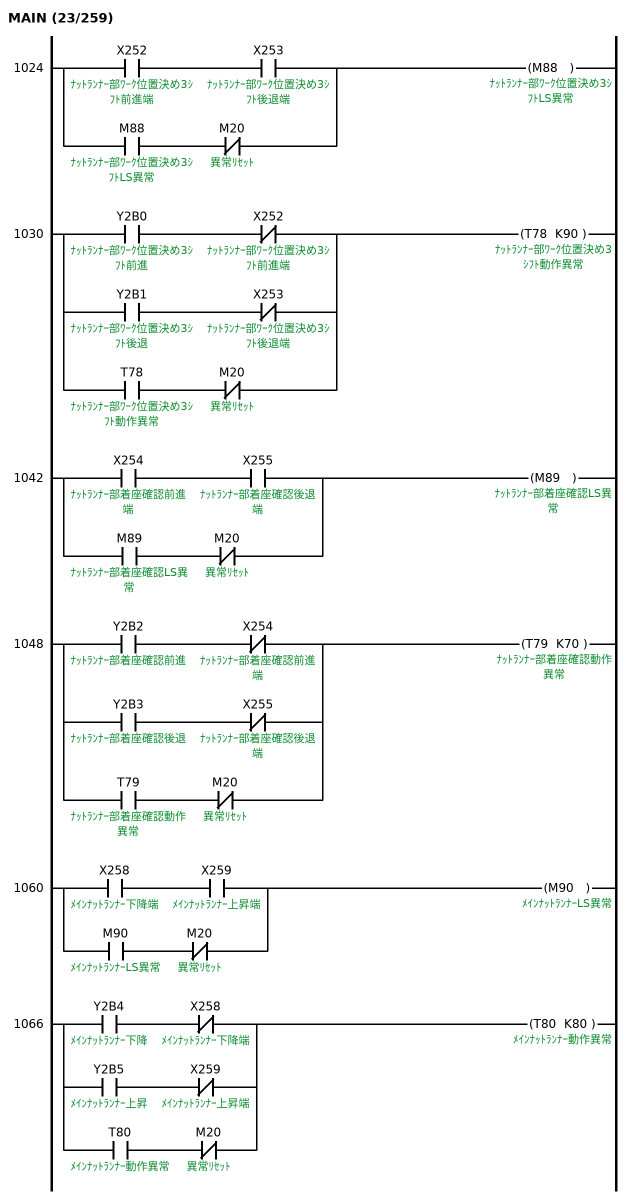
1024  LD      X252  ; ﾅｯﾄﾗﾝﾅｰ部ﾜｰｸ位置決め3ｼﾌﾄ前進端
      AND     X253  ; ﾅｯﾄﾗﾝﾅｰ部ﾜｰｸ位置決め3ｼﾌﾄ後退端
      LD      M88  ; ﾅｯﾄﾗﾝﾅｰ部ﾜｰｸ位置決め3ｼﾌﾄLS異常
      ANI     M20  ; 異常ﾘｾｯﾄ
      ORB
      OUT     M88  ; ﾅｯﾄﾗﾝﾅｰ部ﾜｰｸ位置決め3ｼﾌﾄLS異常
1030  LD      Y2B0  ; ﾅｯﾄﾗﾝﾅｰ部ﾜｰｸ位置決め3ｼﾌﾄ前進
      ANI     X252  ; ﾅｯﾄﾗﾝﾅｰ部ﾜｰｸ位置決め3ｼﾌﾄ前進端
      LD      Y2B1  ; ﾅｯﾄﾗﾝﾅｰ部ﾜｰｸ位置決め3ｼﾌﾄ後退
      ANI     X253  ; ﾅｯﾄﾗﾝﾅｰ部ﾜｰｸ位置決め3ｼﾌﾄ後退端
      ORB
      LD      T78  ; ﾅｯﾄﾗﾝﾅｰ部ﾜｰｸ位置決め3ｼﾌﾄ動作異常
      ANI     M20  ; 異常ﾘｾｯﾄ
      ORB
      OUT     T78 K90  ; ﾅｯﾄﾗﾝﾅｰ部ﾜｰｸ位置決め3ｼﾌﾄ動作異常
1042  LD      X254  ; ﾅｯﾄﾗﾝﾅｰ部着座確認前進端
      AND     X255  ; ﾅｯﾄﾗﾝﾅｰ部着座確認後退端
      LD      M89  ; ﾅｯﾄﾗﾝﾅｰ部着座確認LS異常
      ANI     M20  ; 異常ﾘｾｯﾄ
      ORB
      OUT     M89  ; ﾅｯﾄﾗﾝﾅｰ部着座確認LS異常
1048  LD      Y2B2  ; ﾅｯﾄﾗﾝﾅｰ部着座確認前進
      ANI     X254  ; ﾅｯﾄﾗﾝﾅｰ部着座確認前進端
      LD      Y2B3  ; ﾅｯﾄﾗﾝﾅｰ部着座確認後退
      ANI     X255  ; ﾅｯﾄﾗﾝﾅｰ部着座確認後退端
      ORB
      LD      T79  ; ﾅｯﾄﾗﾝﾅｰ部着座確認動作異常
      ANI     M20  ; 異常ﾘｾｯﾄ
      ORB
      OUT     T79 K70  ; ﾅｯﾄﾗﾝﾅｰ部着座確認動作異常
1060  LD      X258  ; ﾒｲﾝﾅｯﾄﾗﾝﾅｰ下降端
      AND     X259  ; ﾒｲﾝﾅｯﾄﾗﾝﾅｰ上昇端
      LD      M90  ; ﾒｲﾝﾅｯﾄﾗﾝﾅｰLS異常
      ANI     M20  ; 異常ﾘｾｯﾄ
      ORB
      OUT     M90  ; ﾒｲﾝﾅｯﾄﾗﾝﾅｰLS異常
1066  LD      Y2B4  ; ﾒｲﾝﾅｯﾄﾗﾝﾅｰ下降
      ANI     X258  ; ﾒｲﾝﾅｯﾄﾗﾝﾅｰ下降端
      LD      Y2B5  ; ﾒｲﾝﾅｯﾄﾗﾝﾅｰ上昇
      ANI     X259  ; ﾒｲﾝﾅｯﾄﾗﾝﾅｰ上昇端
      ORB
      LD      T80  ; ﾒｲﾝﾅｯﾄﾗﾝﾅｰ動作異常
      ANI     M20  ; 異常ﾘｾｯﾄ
      ORB
      OUT     T80 K80  ; ﾒｲﾝﾅｯﾄﾗﾝﾅｰ動作異常
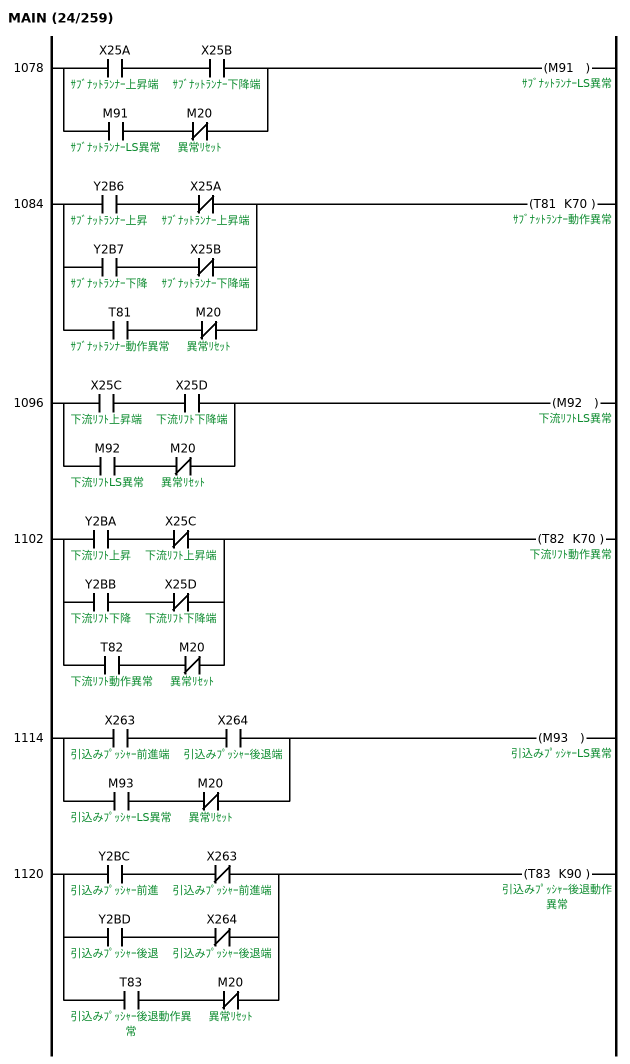
1078  LD      X25A  ; ｻﾌﾞﾅｯﾄﾗﾝﾅｰ上昇端
      AND     X25B  ; ｻﾌﾞﾅｯﾄﾗﾝﾅｰ下降端
      LD      M91  ; ｻﾌﾞﾅｯﾄﾗﾝﾅｰLS異常
      ANI     M20  ; 異常ﾘｾｯﾄ
      ORB
      OUT     M91  ; ｻﾌﾞﾅｯﾄﾗﾝﾅｰLS異常
1084  LD      Y2B6  ; ｻﾌﾞﾅｯﾄﾗﾝﾅｰ上昇
      ANI     X25A  ; ｻﾌﾞﾅｯﾄﾗﾝﾅｰ上昇端
      LD      Y2B7  ; ｻﾌﾞﾅｯﾄﾗﾝﾅｰ下降
      ANI     X25B  ; ｻﾌﾞﾅｯﾄﾗﾝﾅｰ下降端
      ORB
      LD      T81  ; ｻﾌﾞﾅｯﾄﾗﾝﾅｰ動作異常
      ANI     M20  ; 異常ﾘｾｯﾄ
      ORB
      OUT     T81 K70  ; ｻﾌﾞﾅｯﾄﾗﾝﾅｰ動作異常
1096  LD      X25C  ; 下流ﾘﾌﾄ上昇端
      AND     X25D  ; 下流ﾘﾌﾄ下降端
      LD      M92  ; 下流ﾘﾌﾄLS異常
      ANI     M20  ; 異常ﾘｾｯﾄ
      ORB
      OUT     M92  ; 下流ﾘﾌﾄLS異常
1102  LD      Y2BA  ; 下流ﾘﾌﾄ上昇
      ANI     X25C  ; 下流ﾘﾌﾄ上昇端
      LD      Y2BB  ; 下流ﾘﾌﾄ下降
      ANI     X25D  ; 下流ﾘﾌﾄ下降端
      ORB
      LD      T82  ; 下流ﾘﾌﾄ動作異常
      ANI     M20  ; 異常ﾘｾｯﾄ
      ORB
      OUT     T82 K70  ; 下流ﾘﾌﾄ動作異常
1114  LD      X263  ; 引込みﾌﾟｯｼｬｰ前進端
      AND     X264  ; 引込みﾌﾟｯｼｬｰ後退端
      LD      M93  ; 引込みﾌﾟｯｼｬｰLS異常
      ANI     M20  ; 異常ﾘｾｯﾄ
      ORB
      OUT     M93  ; 引込みﾌﾟｯｼｬｰLS異常
1120  LD      Y2BC  ; 引込みﾌﾟｯｼｬｰ前進
      ANI     X263  ; 引込みﾌﾟｯｼｬｰ前進端
      LD      Y2BD  ; 引込みﾌﾟｯｼｬｰ後退
      ANI     X264  ; 引込みﾌﾟｯｼｬｰ後退端
      ORB
      LD      T83  ; 引込みﾌﾟｯｼｬｰ後退動作異常
      ANI     M20  ; 異常ﾘｾｯﾄ
      ORB
      OUT     T83 K90  ; 引込みﾌﾟｯｼｬｰ後退動作異常
